LIN {X 0,Y 353.137,Z 586.014,A -85,B 0,C 180,E1 15983.414,E2 15983.414} C_VEL
LIN {X 0,Y 345.112,Z 562.488,A -85,B 0,C 180,E1 15988.238,E2 15988.238} C_VEL
LIN {X 0,Y 335.464,Z 541.503,A -85,B 0,C 180,E1 15993.705,E2 15993.705} C_VEL
LIN {X 0,Y 327.139,Z 526.718,A -85,B 0,C 180,E1 15998.911,E2 15998.911} C_VEL
LIN {X 0,Y 320.283,Z 515.167,A -85,B 0,C 180,E1 16004.452,E2 16004.452} C_VEL
LIN {X 0,Y 316.039,Z 508.566,A -85,B 0,C 180,E1 16009.304,E2 16009.304} C_VEL
LIN {X 0,Y 313.178,Z 504.462,A -85,B 0,C 180,E1 16018.617,E2 16018.617} C_VEL
LIN {X 0,Y 316.834,Z 509.857,A -85,B 0,C 180,E1 16027.466,E2 16027.466} C_VEL
LIN {X 0,Y 321.627,Z 517.983,A -85,B 0,C 180,E1 16032.576,E2 16032.576} C_VEL
LIN {X 0,Y 328.52,Z 529.301,A -85,B 0,C 180,E1 16037.778,E2 16037.778} C_VEL
LIN {X 0,Y 337.694,Z 547.182,A -85,B 0,C 180,E1 16043.535,E2 16043.535} C_VEL
LIN {X 0,Y 346.598,Z 568.688,A -85,B 0,C 180,E1 16048.719,E2 16048.719} C_VEL
LIN {X 0,Y 352.614,Z 590.285,A -85,B 0,C 180,E1 16052.83,E2 16052.83} C_VEL
LIN {X 0,Y 340.82,Z 629.242,A -85,B 0,C 180,E1 16055.81,E2 16055.81} C_VEL
LIN {X 0,Y 327.37,Z 665.336,A -85,B 0,C 180,E1 16059.799,E2 16059.799} C_VEL
LIN {X 0,Y 313.918,Z 696.935,A -85,B 0,C 180,E1 16064.711,E2 16064.711} C_VEL
LIN {X 0,Y 301.373,Z 724.654,A -85,B 0,C 180,E1 16070.701,E2 16070.701} C_VEL
LIN {X 0,Y 290.781,Z 748.154,A -85,B 0,C 180,E1 16077.768,E2 16077.768} C_VEL
LIN {X 0,Y 283.432,Z 766.757,A -85,B 0,C 180,E1 16085.741,E2 16085.741} C_VEL
LIN {X 0,Y 279.612,Z 780.048,A -85,B 0,C 180,E1 16094.291,E2 16094.291} C_VEL
LIN {X 0,Y 278.455,Z 786.164,A -85,B 0,C 180,E1 16100.611,E2 16100.611} C_VEL
LIN {X 0,Y 278.297,Z 789.212,A -85,B 0,C 180,E1 16106.881,E2 16106.881} C_VEL
LIN {X 0,Y 278.243,Z 789.212,A -85,B 0,C 180,E1 16113.119,E2 16113.119} C_VEL
LIN {X 0,Y 278.634,Z 785.021,A -85,B 0,C 180,E1 16120.802,E2 16120.802} C_VEL
LIN {X 0,Y 280.671,Z 775.811,A -85,B 0,C 180,E1 16128.886,E2 16128.886} C_VEL
LIN {X 0,Y 285.353,Z 761.575,A -85,B 0,C 180,E1 16136.809,E2 16136.809} C_VEL
LIN {X 0,Y 294.373,Z 740.19,A -85,B 0,C 180,E1 16144.905,E2 16144.905} C_VEL
LIN {X 0,Y 306.704,Z 712.859,A -85,B 0,C 180,E1 16152.112,E2 16152.112} C_VEL
LIN {X 0,Y 320.536,Z 682.014,A -85,B 0,C 180,E1 16157.82,E2 16157.82} C_VEL
LIN {X 0,Y 334.611,Z 647.007,A -85,B 0,C 180,E1 16162.409,E2 16162.409} C_VEL
LIN {X 0,Y 347.053,Z 610.454,A -85,B 0,C 180,E1 16165.773,E2 16165.773} C_VEL
LIN {X 0,Y 348.409,Z 599.608,A -85,B 0,C 180,E1 16166.985,E2 16166.985} C_VEL
LIN {X 0,Y 345.391,Z 584.533,A -85,B 0,C 180,E1 16169.727,E2 16169.727} C_VEL
LIN {X 0,Y 337.684,Z 561.735,A -85,B 0,C 180,E1 16174.828,E2 16174.828} C_VEL
LIN {X 0,Y 328.702,Z 541.555,A -85,B 0,C 180,E1 16180.754,E2 16180.754} C_VEL
LIN {X 0,Y 321.259,Z 528.092,A -85,B 0,C 180,E1 16186.457,E2 16186.457} C_VEL
LIN {X 0,Y 317.544,Z 522.011,A -85,B 0,C 180,E1 16190.046,E2 16190.046} C_VEL
LIN {X 0,Y 314.711,Z 516.201,A -85,B 0,C 180,E1 16194.131,E2 16194.131} C_VEL
LIN {X 0,Y 312.367,Z 513.05,A -85,B 0,C 180,E1 16199.998,E2 16199.998} C_VEL
LIN {X 0,Y 312.759,Z 514.467,A -85,B 0,C 180,E1 16206.251,E2 16206.251} C_VEL
LIN {X 0,Y 315.457,Z 517.712,A -85,B 0,C 180,E1 16211.31,E2 16211.31} C_VEL
LIN {X 0,Y 319.83,Z 525.512,A -85,B 0,C 180,E1 16216.411,E2 16216.411} C_VEL
LIN {X 0,Y 326.074,Z 535.896,A -85,B 0,C 180,E1 16221.437,E2 16221.437} C_VEL
LIN {X 0,Y 335.111,Z 553.88,A -85,B 0,C 180,E1 16227.401,E2 16227.401} C_VEL
LIN {X 0,Y 343.589,Z 575.487,A -85,B 0,C 180,E1 16232.717,E2 16232.717} C_VEL
LIN {X 0,Y 347.738,Z 591.04,A -85,B 0,C 180,E1 16235.805,E2 16235.805} C_VEL
LIN {X 0,Y 336.302,Z 626.527,A -85,B 0,C 180,E1 16238.531,E2 16238.531} C_VEL
LIN {X 0,Y 323.487,Z 658.718,A -85,B 0,C 180,E1 16242.125,E2 16242.125} C_VEL
LIN {X 0,Y 309.543,Z 688.272,A -85,B 0,C 180,E1 16246.779,E2 16246.779} C_VEL
LIN {X 0,Y 296.072,Z 714.128,A -85,B 0,C 180,E1 16252.606,E2 16252.606} C_VEL
LIN {X 0,Y 284.563,Z 735.641,A -85,B 0,C 180,E1 16259.636,E2 16259.636} C_VEL
LIN {X 0,Y 276.615,Z 751.803,A -85,B 0,C 180,E1 16267.47,E2 16267.47} C_VEL
LIN {X 0,Y 272.314,Z 762.47,A -85,B 0,C 180,E1 16275.51,E2 16275.51} C_VEL
LIN {X 0,Y 270.547,Z 768.232,A -85,B 0,C 180,E1 16283.573,E2 16283.573} C_VEL
LIN {X 0,Y 270.584,Z 769.634,A -85,B 0,C 180,E1 16290,E2 16290} C_VEL
LIN {X 0,Y 270.553,Z 768.178,A -85,B 0,C 180,E1 16296.427,E2 16296.427} C_VEL
LIN {X 0,Y 272.343,Z 762.375,A -85,B 0,C 180,E1 16304.489,E2 16304.489} C_VEL
LIN {X 0,Y 277.243,Z 750.314,A -85,B 0,C 180,E1 16313.325,E2 16313.325} C_VEL
LIN {X 0,Y 286.184,Z 732.442,A -85,B 0,C 180,E1 16321.498,E2 16321.498} C_VEL
LIN {X 0,Y 297.829,Z 710.843,A -85,B 0,C 180,E1 16328.155,E2 16328.155} C_VEL
LIN {X 0,Y 311.444,Z 684.319,A -85,B 0,C 180,E1 16333.851,E2 16333.851} C_VEL
LIN {X 0,Y 325.748,Z 653.106,A -85,B 0,C 180,E1 16338.516,E2 16338.516} C_VEL
LIN {X 0,Y 339.264,Z 617.956,A -85,B 0,C 180,E1 16342.129,E2 16342.129} C_VEL
LIN {X 0,Y 347.721,Z 589.37,A -85,B 0,C 180,E1 16344.295,E2 16344.295} C_VEL
LIN {X 0,Y 339.611,Z 564.718,A -85,B 0,C 180,E1 16349.644,E2 16349.644} C_VEL
LIN {X 0,Y 330.372,Z 544.154,A -85,B 0,C 180,E1 16355.464,E2 16355.464} C_VEL
LIN {X 0,Y 322.011,Z 528.726,A -85,B 0,C 180,E1 16361.536,E2 16361.536} C_VEL
LIN {X 0,Y 317.486,Z 521.686,A -85,B 0,C 180,E1 16365.708,E2 16365.708} C_VEL
LIN {X 0,Y 314.63,Z 516.234,A -85,B 0,C 180,E1 16369.65,E2 16369.65} C_VEL
LIN {X 0,Y 312.04,Z 512.261,A -85,B 0,C 180,E1 16378.611,E2 16378.611} C_VEL
LIN {X 0,Y 315.364,Z 517.62,A -85,B 0,C 180,E1 16387.241,E2 16387.241} C_VEL
LIN {X 0,Y 319.799,Z 525.722,A -85,B 0,C 180,E1 16392.388,E2 16392.388} C_VEL
LIN {X 0,Y 325.91,Z 536.494,A -85,B 0,C 180,E1 16397.402,E2 16397.402} C_VEL
LIN {X 0,Y 334.33,Z 553.843,A -85,B 0,C 180,E1 16403.098,E2 16403.098} C_VEL
LIN {X 0,Y 342.861,Z 576.373,A -85,B 0,C 180,E1 16408.609,E2 16408.609} C_VEL
LIN {X 0,Y 347.106,Z 593.898,A -85,B 0,C 180,E1 16411.983,E2 16411.983} C_VEL
LIN {X 0,Y 335.107,Z 631.506,A -85,B 0,C 180,E1 16414.94,E2 16414.94} C_VEL
LIN {X 0,Y 321.819,Z 665.824,A -85,B 0,C 180,E1 16418.808,E2 16418.808} C_VEL
LIN {X 0,Y 308.231,Z 696.335,A -85,B 0,C 180,E1 16423.57,E2 16423.57} C_VEL
LIN {X 0,Y 294.83,Z 724.689,A -85,B 0,C 180,E1 16429.787,E2 16429.787} C_VEL
LIN {X 0,Y 283.811,Z 747.971,A -85,B 0,C 180,E1 16436.937,E2 16436.937} C_VEL
LIN {X 0,Y 276.045,Z 766.29,A -85,B 0,C 180,E1 16444.966,E2 16444.966} C_VEL
LIN {X 0,Y 271.827,Z 779.746,A -85,B 0,C 180,E1 16453.829,E2 16453.829} C_VEL
LIN {X 0,Y 270.574,Z 785.87,A -85,B 0,C 180,E1 16460.335,E2 16460.335} C_VEL
LIN {X 0,Y 270.401,Z 788.924,A -85,B 0,C 180,E1 16466.79,E2 16466.79} C_VEL
LIN {X 0,Y 270.355,Z 788.925,A -85,B 0,C 180,E1 16473.21,E2 16473.21} C_VEL
LIN {X 0,Y 270.774,Z 784.86,A -85,B 0,C 180,E1 16480.953,E2 16480.953} C_VEL
LIN {X 0,Y 273,Z 775.452,A -85,B 0,C 180,E1 16489.476,E2 16489.476} C_VEL
LIN {X 0,Y 278.038,Z 761.26,A -85,B 0,C 180,E1 16497.574,E2 16497.574} C_VEL
LIN {X 0,Y 287.656,Z 739.855,A -85,B 0,C 180,E1 16505.844,E2 16505.844} C_VEL
LIN {X 0,Y 300.675,Z 712.5,A -85,B 0,C 180,E1 16513.159,E2 16513.159} C_VEL
LIN {X 0,Y 315.05,Z 681.606,A -85,B 0,C 180,E1 16518.933,E2 16518.933} C_VEL
LIN {X 0,Y 329.561,Z 646.887,A -85,B 0,C 180,E1 16523.495,E2 16523.495} C_VEL
LIN {X 0,Y 342.623,Z 609.563,A -85,B 0,C 180,E1 16526.92,E2 16526.92} C_VEL
LIN {X 0,Y 347.405,Z 592.925,A -85,B 0,C 180,E1 16528.102,E2 16528.102} C_VEL
LIN {X 0,Y 345.391,Z 584.533,A -85,B 0,C 180,E1 16529.727,E2 16529.727} C_VEL
LIN {X 0,Y 341.684,Z 578.36,A -85,B 0,C 180,E1 16531.557,E2 16531.557} C_VEL
LIN {X 0,Y 334.557,Z 569.967,A -85,B 0,C 180,E1 16534.821,E2 16534.821} C_VEL
LIN {X 0,Y 326.525,Z 550.443,A -85,B 0,C 180,E1 16540.532,E2 16540.532} C_VEL
LIN {X 0,Y 319.453,Z 536.042,A -85,B 0,C 180,E1 16546.379,E2 16546.379} C_VEL
LIN {X 0,Y 315.565,Z 529.312,A -85,B 0,C 180,E1 16550.506,E2 16550.506} C_VEL
LIN {X 0,Y 312.771,Z 523.658,A -85,B 0,C 180,E1 16554.791,E2 16554.791} C_VEL
LIN {X 0,Y 310.987,Z 520.863,A -85,B 0,C 180,E1 16559.998,E2 16559.998} C_VEL
LIN {X 0,Y 311.369,Z 522.333,A -85,B 0,C 180,E1 16566.371,E2 16566.371} C_VEL
LIN {X 0,Y 313.758,Z 525.368,A -85,B 0,C 180,E1 16571.064,E2 16571.064} C_VEL
LIN {X 0,Y 317.849,Z 533.119,A -85,B 0,C 180,E1 16576.165,E2 16576.165} C_VEL
LIN {X 0,Y 323.837,Z 543.834,A -85,B 0,C 180,E1 16581.317,E2 16581.317} C_VEL
LIN {X 0,Y 331.922,Z 561.078,A -85,B 0,C 180,E1 16587.135,E2 16587.135} C_VEL
LIN {X 0,Y 339.909,Z 583.609,A -85,B 0,C 180,E1 16592.711,E2 16592.711} C_VEL
LIN {X 0,Y 342.528,Z 593.61,A -85,B 0,C 180,E1 16594.827,E2 16594.827} C_VEL
LIN {X 0,Y 329.727,Z 631.56,A -85,B 0,C 180,E1 16597.883,E2 16597.883} C_VEL
LIN {X 0,Y 314.704,Z 666.624,A -85,B 0,C 180,E1 16602.078,E2 16602.078} C_VEL
LIN {X 0,Y 299.679,Z 696.377,A -85,B 0,C 180,E1 16607.288,E2 16607.288} C_VEL
LIN {X 0,Y 285.425,Z 722.099,A -85,B 0,C 180,E1 16613.879,E2 16613.879} C_VEL
LIN {X 0,Y 274.858,Z 741.051,A -85,B 0,C 180,E1 16620.971,E2 16620.971} C_VEL
LIN {X 0,Y 267.351,Z 755.919,A -85,B 0,C 180,E1 16629.316,E2 16629.316} C_VEL
LIN {X 0,Y 263.877,Z 764.691,A -85,B 0,C 180,E1 16637.243,E2 16637.243} C_VEL
LIN {X 0,Y 262.664,Z 768.521,A -85,B 0,C 180,E1 16643.38,E2 16643.38} C_VEL
LIN {X 0,Y 262.684,Z 769.921,A -85,B 0,C 180,E1 16650,E2 16650} C_VEL
LIN {X 0,Y 262.671,Z 768.468,A -85,B 0,C 180,E1 16656.62,E2 16656.62} C_VEL
LIN {X 0,Y 264.602,Z 762.668,A -85,B 0,C 180,E1 16664.922,E2 16664.922} C_VEL
LIN {X 0,Y 269.839,Z 750.62,A -85,B 0,C 180,E1 16674.005,E2 16674.005} C_VEL
LIN {X 0,Y 279.318,Z 732.761,A -85,B 0,C 180,E1 16682.365,E2 16682.365} C_VEL
LIN {X 0,Y 292.134,Z 710.066,A -85,B 0,C 180,E1 16689.414,E2 16689.414} C_VEL
LIN {X 0,Y 306.658,Z 682.818,A -85,B 0,C 180,E1 16695.216,E2 16695.216} C_VEL
LIN {X 0,Y 321.286,Z 651.843,A -85,B 0,C 180,E1 16699.78,E2 16699.78} C_VEL
LIN {X 0,Y 335.034,Z 616.822,A -85,B 0,C 180,E1 16703.339,E2 16703.339} C_VEL
LIN {X 0,Y 342.454,Z 593.221,A -85,B 0,C 180,E1 16705.119,E2 16705.119} C_VEL
LIN {X 0,Y 335.089,Z 569.345,A -85,B 0,C 180,E1 16710.535,E2 16710.535} C_VEL
LIN {X 0,Y 326.861,Z 550.145,A -85,B 0,C 180,E1 16716.184,E2 16716.184} C_VEL
LIN {X 0,Y 319.519,Z 535.81,A -85,B 0,C 180,E1 16722.045,E2 16722.045} C_VEL
LIN {X 0,Y 315.478,Z 528.945,A -85,B 0,C 180,E1 16726.216,E2 16726.216} C_VEL
LIN {X 0,Y 312.922,Z 523.837,A -85,B 0,C 180,E1 16729.968,E2 16729.968} C_VEL
LIN {X 0,Y 310.706,Z 520.048,A -85,B 0,C 180,E1 16738.606,E2 16738.606} C_VEL
LIN {X 0,Y 313.615,Z 525.144,A -85,B 0,C 180,E1 16746.933,E2 16746.933} C_VEL
LIN {X 0,Y 317.885,Z 533.565,A -85,B 0,C 180,E1 16752.29,E2 16752.29} C_VEL
LIN {X 0,Y 323.985,Z 545.148,A -85,B 0,C 180,E1 16757.592,E2 16757.592} C_VEL
LIN {X 0,Y 331.143,Z 561.142,A -85,B 0,C 180,E1 16762.861,E2 16762.861} C_VEL
LIN {X 0,Y 338.456,Z 582.174,A -85,B 0,C 180,E1 16768.102,E2 16768.102} C_VEL
LIN {X 0,Y 341.793,Z 597.172,A -85,B 0,C 180,E1 16771.093,E2 16771.093} C_VEL
LIN {X 0,Y 327.694,Z 638.464,A -85,B 0,C 180,E1 16774.49,E2 16774.49} C_VEL
LIN {X 0,Y 312.596,Z 674.634,A -85,B 0,C 180,E1 16778.92,E2 16778.92} C_VEL
LIN {X 0,Y 297.477,Z 706.575,A -85,B 0,C 180,E1 16784.554,E2 16784.554} C_VEL
LIN {X 0,Y 283.977,Z 733.239,A -85,B 0,C 180,E1 16791.208,E2 16791.208} C_VEL
LIN {X 0,Y 272.971,Z 755.957,A -85,B 0,C 180,E1 16799.373,E2 16799.373} C_VEL
LIN {X 0,Y 266.107,Z 772.766,A -85,B 0,C 180,E1 16808.294,E2 16808.294} C_VEL
LIN {X 0,Y 263.218,Z 782.902,A -85,B 0,C 180,E1 16816.697,E2 16816.697} C_VEL
LIN {X 0,Y 262.421,Z 787.482,A -85,B 0,C 180,E1 16823.373,E2 16823.373} C_VEL
LIN {X 0,Y 262.646,Z 789.025,A -85,B 0,C 180,E1 16830,E2 16830} C_VEL
LIN {X 0,Y 262.426,Z 787.489,A -85,B 0,C 180,E1 16836.626,E2 16836.626} C_VEL
LIN {X 0,Y 263.606,Z 781.259,A -85,B 0,C 180,E1 16844.98,E2 16844.98} C_VEL
LIN {X 0,Y 267.024,Z 770.117,A -85,B 0,C 180,E1 16853.386,E2 16853.386} C_VEL
LIN {X 0,Y 274.247,Z 753.319,A -85,B 0,C 180,E1 16861.755,E2 16861.755} C_VEL
LIN {X 0,Y 285.355,Z 730.673,A -85,B 0,C 180,E1 16869.549,E2 16869.549} C_VEL
LIN {X 0,Y 299.435,Z 702.663,A -85,B 0,C 180,E1 16876.269,E2 16876.269} C_VEL
LIN {X 0,Y 314.667,Z 670.229,A -85,B 0,C 180,E1 16881.715,E2 16881.715} C_VEL
LIN {X 0,Y 329.211,Z 634.734,A -85,B 0,C 180,E1 16885.881,E2 16885.881} C_VEL
LIN {X 0,Y 342.019,Z 596.191,A -85,B 0,C 180,E1 16889.016,E2 16889.016} C_VEL
LIN {X 0,Y 335.616,Z 572.905,A -85,B 0,C 180,E1 16894.076,E2 16894.076} C_VEL
LIN {X 0,Y 334.557,Z 569.967,A -85,B 0,C 180,E1 16894.821,E2 16894.821} C_VEL
LIN {X 0,Y 330.732,Z 565.067,A -85,B 0,C 180,E1 16896.813,E2 16896.813} C_VEL
LIN {X 0,Y 324.612,Z 559.901,A -85,B 0,C 180,E1 16900.015,E2 16900.015} C_VEL
LIN {X 0,Y 324.191,Z 558.921,A -85,B 0,C 180,E1 16900.358,E2 16900.358} C_VEL
LIN {X 0,Y 317.096,Z 543.325,A -85,B 0,C 180,E1 16906.721,E2 16906.721} C_VEL
LIN {X 0,Y 313.157,Z 536.373,A -85,B 0,C 180,E1 16911.134,E2 16911.134} C_VEL
LIN {X 0,Y 311.193,Z 531.423,A -85,B 0,C 180,E1 16914.765,E2 16914.765} C_VEL
LIN {X 0,Y 309.487,Z 528.638,A -85,B 0,C 180,E1 16919.998,E2 16919.998} C_VEL
LIN {X 0,Y 309.811,Z 530.002,A -85,B 0,C 180,E1 16926.189,E2 16926.189} C_VEL
LIN {X 0,Y 311.916,Z 532.916,A -85,B 0,C 180,E1 16930.77,E2 16930.77} C_VEL
LIN {X 0,Y 315.728,Z 540.724,A -85,B 0,C 180,E1 16935.978,E2 16935.978} C_VEL
LIN {X 0,Y 321.027,Z 551.025,A -85,B 0,C 180,E1 16940.983,E2 16940.983} C_VEL
LIN {X 0,Y 328.008,Z 566.848,A -85,B 0,C 180,E1 16946.464,E2 16946.464} C_VEL
LIN {X 0,Y 335.297,Z 589.367,A -85,B 0,C 180,E1 16952.222,E2 16952.222} C_VEL
LIN {X 0,Y 336.939,Z 598.552,A -85,B 0,C 180,E1 16954.062,E2 16954.062} C_VEL
LIN {X 0,Y 323.756,Z 634.87,A -85,B 0,C 180,E1 16957.063,E2 16957.063} C_VEL
LIN {X 0,Y 308.734,Z 668.307,A -85,B 0,C 180,E1 16961.174,E2 16961.174} C_VEL
LIN {X 0,Y 293.399,Z 697.437,A -85,B 0,C 180,E1 16966.381,E2 16966.381} C_VEL
LIN {X 0,Y 279.454,Z 721.6,A -85,B 0,C 180,E1 16972.64,E2 16972.64} C_VEL
LIN {X 0,Y 267.915,Z 741.21,A -85,B 0,C 180,E1 16980.062,E2 16980.062} C_VEL
LIN {X 0,Y 259.727,Z 756.417,A -85,B 0,C 180,E1 16988.845,E2 16988.845} C_VEL
LIN {X 0,Y 256.244,Z 764.534,A -85,B 0,C 180,E1 16996.328,E2 16996.328} C_VEL
LIN {X 0,Y 254.782,Z 768.809,A -85,B 0,C 180,E1 17003.174,E2 17003.174} C_VEL
LIN {X 0,Y 254.802,Z 770.208,A -85,B 0,C 180,E1 17010,E2 17010} C_VEL
LIN {X 0,Y 254.79,Z 768.757,A -85,B 0,C 180,E1 17016.826,E2 17016.826} C_VEL
LIN {X 0,Y 256.851,Z 762.961,A -85,B 0,C 180,E1 17025.383,E2 17025.383} C_VEL
LIN {X 0,Y 262.503,Z 750.924,A -85,B 0,C 180,E1 17034.72,E2 17034.72} C_VEL
LIN {X 0,Y 272.538,Z 733.077,A -85,B 0,C 180,E1 17043.273,E2 17043.273} C_VEL
LIN {X 0,Y 285.949,Z 710.405,A -85,B 0,C 180,E1 17050.44,E2 17050.44} C_VEL
LIN {X 0,Y 301.066,Z 683.188,A -85,B 0,C 180,E1 17056.299,E2 17056.299} C_VEL
LIN {X 0,Y 316.129,Z 652.423,A -85,B 0,C 180,E1 17060.866,E2 17060.866} C_VEL
LIN {X 0,Y 330.369,Z 617.365,A -85,B 0,C 180,E1 17064.441,E2 17064.441} C_VEL
LIN {X 0,Y 337.064,Z 597.828,A -85,B 0,C 180,E1 17065.891,E2 17065.891} C_VEL
LIN {X 0,Y 332.03,Z 578.634,A -85,B 0,C 180,E1 17070.237,E2 17070.237} C_VEL
LIN {X 0,Y 324.684,Z 558.924,A -85,B 0,C 180,E1 17075.922,E2 17075.922} C_VEL
LIN {X 0,Y 317.28,Z 543.256,A -85,B 0,C 180,E1 17082.301,E2 17082.301} C_VEL
LIN {X 0,Y 313.251,Z 536.151,A -85,B 0,C 180,E1 17086.702,E2 17086.702} C_VEL
LIN {X 0,Y 311.15,Z 531.459,A -85,B 0,C 180,E1 17090.286,E2 17090.286} C_VEL
LIN {X 0,Y 309.213,Z 527.806,A -85,B 0,C 180,E1 17098.599,E2 17098.599} C_VEL
LIN {X 0,Y 311.766,Z 532.824,A -85,B 0,C 180,E1 17106.712,E2 17106.712} C_VEL
LIN {X 0,Y 315.732,Z 541.197,A -85,B 0,C 180,E1 17112.111,E2 17112.111} C_VEL
LIN {X 0,Y 322.296,Z 554.591,A -85,B 0,C 180,E1 17118.19,E2 17118.19} C_VEL
LIN {X 0,Y 330.026,Z 574.809,A -85,B 0,C 180,E1 17124.386,E2 17124.386} C_VEL
LIN {X 0,Y 336.228,Z 597.696,A -85,B 0,C 180,E1 17129.691,E2 17129.691} C_VEL
LIN {X 0,Y 335.819,Z 602.485,A -85,B 0,C 180,E1 17130.332,E2 17130.332} C_VEL
LIN {X 0,Y 322.438,Z 639.685,A -85,B 0,C 180,E1 17133.474,E2 17133.474} C_VEL
LIN {X 0,Y 306.978,Z 675.305,A -85,B 0,C 180,E1 17137.891,E2 17137.891} C_VEL
LIN {X 0,Y 291.715,Z 706.212,A -85,B 0,C 180,E1 17143.392,E2 17143.392} C_VEL
LIN {X 0,Y 277.403,Z 733.23,A -85,B 0,C 180,E1 17150.24,E2 17150.24} C_VEL
LIN {X 0,Y 266.226,Z 755.026,A -85,B 0,C 180,E1 17158.185,E2 17158.185} C_VEL
LIN {X 0,Y 258.962,Z 771.185,A -85,B 0,C 180,E1 17166.755,E2 17166.755} C_VEL
LIN {X 0,Y 255.816,Z 780.95,A -85,B 0,C 180,E1 17174.553,E2 17174.553} C_VEL
LIN {X 0,Y 254.537,Z 787.192,A -85,B 0,C 180,E1 17183.167,E2 17183.167} C_VEL
LIN {X 0,Y 254.768,Z 788.739,A -85,B 0,C 180,E1 17190,E2 17190} C_VEL
LIN {X 0,Y 254.542,Z 787.199,A -85,B 0,C 180,E1 17196.833,E2 17196.833} C_VEL
LIN {X 0,Y 255.815,Z 780.963,A -85,B 0,C 180,E1 17205.447,E2 17205.447} C_VEL
LIN {X 0,Y 259.513,Z 769.809,A -85,B 0,C 180,E1 17214.105,E2 17214.105} C_VEL
LIN {X 0,Y 267.13,Z 753.13,A -85,B 0,C 180,E1 17222.64,E2 17222.64} C_VEL
LIN {X 0,Y 279.006,Z 730.332,A -85,B 0,C 180,E1 17230.634,E2 17230.634} C_VEL
LIN {X 0,Y 293.95,Z 701.944,A -85,B 0,C 180,E1 17237.504,E2 17237.504} C_VEL
LIN {X 0,Y 309.645,Z 669.808,A -85,B 0,C 180,E1 17242.908,E2 17242.908} C_VEL
LIN {X 0,Y 324.741,Z 634.232,A -85,B 0,C 180,E1 17247.063,E2 17247.063} C_VEL
LIN {X 0,Y 336.639,Z 599.376,A -85,B 0,C 180,E1 17249.978,E2 17249.978} C_VEL
LIN {X 0,Y 331.372,Z 578.764,A -85,B 0,C 180,E1 17254.618,E2 17254.618} C_VEL
LIN {X 0,Y 324.191,Z 558.921,A -85,B 0,C 180,E1 17260.358,E2 17260.358} C_VEL
LIN {X 0,Y 320.766,Z 555.603,A -85,B 0,C 180,E1 17262.536,E2 17262.536} C_VEL
LIN {X 0,Y 315.39,Z 552.897,A -85,B 0,C 180,E1 17265.975,E2 17265.975} C_VEL
LIN {X 0,Y 315.066,Z 552.056,A -85,B 0,C 180,E1 17266.343,E2 17266.343} C_VEL
LIN {X 0,Y 311.27,Z 544.188,A -85,B 0,C 180,E1 17271.08,E2 17271.08} C_VEL
LIN {X 0,Y 308.977,Z 538.755,A -85,B 0,C 180,E1 17275.432,E2 17275.432} C_VEL
LIN {X 0,Y 307.692,Z 536.354,A -85,B 0,C 180,E1 17279.998,E2 17279.998} C_VEL
LIN {X 0,Y 307.932,Z 537.6,A -85,B 0,C 180,E1 17286.012,E2 17286.012} C_VEL
LIN {X 0,Y 309.883,Z 540.498,A -85,B 0,C 180,E1 17290.522,E2 17290.522} C_VEL
LIN {X 0,Y 313.385,Z 548.242,A -85,B 0,C 180,E1 17295.765,E2 17295.765} C_VEL
LIN {X 0,Y 318.425,Z 558.829,A -85,B 0,C 180,E1 17300.889,E2 17300.889} C_VEL
LIN {X 0,Y 324.355,Z 573.435,A -85,B 0,C 180,E1 17306.039,E2 17306.039} C_VEL
LIN {X 0,Y 330.746,Z 595.28,A -85,B 0,C 180,E1 17311.761,E2 17311.761} C_VEL
LIN {X 0,Y 331.855,Z 601.305,A -85,B 0,C 180,E1 17313.087,E2 17313.087} C_VEL
LIN {X 0,Y 318.442,Z 636.689,A -85,B 0,C 180,E1 17316.068,E2 17316.068} C_VEL
LIN {X 0,Y 303.353,Z 669.041,A -85,B 0,C 180,E1 17320.095,E2 17320.095} C_VEL
LIN {X 0,Y 287.64,Z 697.774,A -85,B 0,C 180,E1 17325.278,E2 17325.278} C_VEL
LIN {X 0,Y 272.876,Z 722.214,A -85,B 0,C 180,E1 17331.707,E2 17331.707} C_VEL
LIN {X 0,Y 260.602,Z 742.052,A -85,B 0,C 180,E1 17339.445,E2 17339.445} C_VEL
LIN {X 0,Y 252.248,Z 756.711,A -85,B 0,C 180,E1 17348.186,E2 17348.186} C_VEL
LIN {X 0,Y 248.01,Z 766.142,A -85,B 0,C 180,E1 17357.599,E2 17357.599} C_VEL
LIN {X 0,Y 246.734,Z 770.155,A -85,B 0,C 180,E1 17366.482,E2 17366.482} C_VEL
LIN {X 0,Y 246.751,Z 770.124,A -85,B 0,C 180,E1 17373.518,E2 17373.518} C_VEL
LIN {X 0,Y 248.033,Z 766.054,A -85,B 0,C 180,E1 17382.425,E2 17382.425} C_VEL
LIN {X 0,Y 252.307,Z 756.528,A -85,B 0,C 180,E1 17391.849,E2 17391.849} C_VEL
LIN {X 0,Y 260.701,Z 741.816,A -85,B 0,C 180,E1 17400.565,E2 17400.565} C_VEL
LIN {X 0,Y 274.092,Z 720.165,A -85,B 0,C 180,E1 17408.846,E2 17408.846} C_VEL
LIN {X 0,Y 289.761,Z 693.948,A -85,B 0,C 180,E1 17415.433,E2 17415.433} C_VEL
LIN {X 0,Y 306.053,Z 663.415,A -85,B 0,C 180,E1 17420.624,E2 17420.624} C_VEL
LIN {X 0,Y 321.023,Z 630.34,A -85,B 0,C 180,E1 17424.45,E2 17424.45} C_VEL
LIN {X 0,Y 331.793,Z 600.108,A -85,B 0,C 180,E1 17426.998,E2 17426.998} C_VEL
LIN {X 0,Y 326.001,Z 578.645,A -85,B 0,C 180,E1 17432.33,E2 17432.33} C_VEL
LIN {X 0,Y 319.718,Z 561.77,A -85,B 0,C 180,E1 17437.741,E2 17437.741} C_VEL
LIN {X 0,Y 313.606,Z 548.705,A -85,B 0,C 180,E1 17443.734,E2 17443.734} C_VEL
LIN {X 0,Y 310.836,Z 543.113,A -85,B 0,C 180,E1 17447.395,E2 17447.395} C_VEL
LIN {X 0,Y 309.044,Z 538.926,A -85,B 0,C 180,E1 17450.724,E2 17450.724} C_VEL
LIN {X 0,Y 307.469,Z 535.482,A -85,B 0,C 180,E1 17458.591,E2 17458.591} C_VEL
LIN {X 0,Y 309.742,Z 540.392,A -85,B 0,C 180,E1 17466.492,E2 17466.492} C_VEL
LIN {X 0,Y 313.817,Z 549.6,A -85,B 0,C 180,E1 17472.452,E2 17472.452} C_VEL
LIN {X 0,Y 319.405,Z 562.422,A -85,B 0,C 180,E1 17478.089,E2 17478.089} C_VEL
LIN {X 0,Y 326.051,Z 581.254,A -85,B 0,C 180,E1 17483.974,E2 17483.974} C_VEL
LIN {X 0,Y 331.097,Z 601.956,A -85,B 0,C 180,E1 17488.936,E2 17488.936} C_VEL
LIN {X 0,Y 330.348,Z 606.289,A -85,B 0,C 180,E1 17489.442,E2 17489.442} C_VEL
LIN {X 0,Y 316.103,Z 643.756,A -85,B 0,C 180,E1 17492.728,E2 17492.728} C_VEL
LIN {X 0,Y 300.57,Z 677.734,A -85,B 0,C 180,E1 17497.088,E2 17497.088} C_VEL
LIN {X 0,Y 285.259,Z 707.355,A -85,B 0,C 180,E1 17502.519,E2 17502.519} C_VEL
LIN {X 0,Y 270.314,Z 734.237,A -85,B 0,C 180,E1 17509.549,E2 17509.549} C_VEL
LIN {X 0,Y 259.122,Z 754.847,A -85,B 0,C 180,E1 17517.282,E2 17517.282} C_VEL
LIN {X 0,Y 251.438,Z 770.875,A -85,B 0,C 180,E1 17526.016,E2 17526.016} C_VEL
LIN {X 0,Y 248.035,Z 780.653,A -85,B 0,C 180,E1 17534.056,E2 17534.056} C_VEL
LIN {X 0,Y 246.632,Z 786.901,A -85,B 0,C 180,E1 17542.947,E2 17542.947} C_VEL
LIN {X 0,Y 246.866,Z 788.451,A -85,B 0,C 180,E1 17550,E2 17550} C_VEL
LIN {X 0,Y 246.638,Z 786.909,A -85,B 0,C 180,E1 17557.053,E2 17557.053} C_VEL
LIN {X 0,Y 248.034,Z 780.667,A -85,B 0,C 180,E1 17565.944,E2 17565.944} C_VEL
LIN {X 0,Y 252.036,Z 769.502,A -85,B 0,C 180,E1 17574.868,E2 17574.868} C_VEL
LIN {X 0,Y 260.107,Z 752.936,A -85,B 0,C 180,E1 17583.574,E2 17583.574} C_VEL
LIN {X 0,Y 272.793,Z 729.994,A -85,B 0,C 180,E1 17591.764,E2 17591.764} C_VEL
LIN {X 0,Y 288.133,Z 702.186,A -85,B 0,C 180,E1 17598.589,E2 17598.589} C_VEL
LIN {X 0,Y 304.219,Z 670.568,A -85,B 0,C 180,E1 17603.977,E2 17603.977} C_VEL
LIN {X 0,Y 319.79,Z 635.289,A -85,B 0,C 180,E1 17608.136,E2 17608.136} C_VEL
LIN {X 0,Y 331.398,Z 603.562,A -85,B 0,C 180,E1 17610.751,E2 17610.751} C_VEL
LIN {X 0,Y 326.346,Z 582.066,A -85,B 0,C 180,E1 17615.851,E2 17615.851} C_VEL
LIN {X 0,Y 319.397,Z 562.07,A -85,B 0,C 180,E1 17622.066,E2 17622.066} C_VEL
LIN {X 0,Y 315.066,Z 552.056,A -85,B 0,C 180,E1 17626.343,E2 17626.343} C_VEL
LIN {X 0,Y 313.118,Z 551.062,A -85,B 0,C 180,E1 17627.879,E2 17627.879} C_VEL
LIN {X 0,Y 309.401,Z 552.394,A -85,B 0,C 180,E1 17630.566,E2 17630.566} C_VEL
LIN {X 0,Y 306.846,Z 546.241,A -85,B 0,C 180,E1 17635.754,E2 17635.754} C_VEL
LIN {X 0,Y 305.711,Z 543.87,A -85,B 0,C 180,E1 17642.837,E2 17642.837} C_VEL
LIN {X 0,Y 307.702,Z 548.113,A -85,B 0,C 180,E1 17650.347,E2 17650.347} C_VEL
LIN {X 0,Y 311.109,Z 556.094,A -85,B 0,C 180,E1 17655.794,E2 17655.794} C_VEL
LIN {X 0,Y 316.58,Z 568.715,A -85,B 0,C 180,E1 17661.752,E2 17661.752} C_VEL
LIN {X 0,Y 322.564,Z 586.776,A -85,B 0,C 180,E1 17667.6,E2 17667.6} C_VEL
LIN {X 0,Y 326.677,Z 604.352,A -85,B 0,C 180,E1 17672.076,E2 17672.076} C_VEL
LIN {X 0,Y 312.287,Z 640.625,A -85,B 0,C 180,E1 17675.261,E2 17675.261} C_VEL
LIN {X 0,Y 296.493,Z 672.735,A -85,B 0,C 180,E1 17679.43,E2 17679.43} C_VEL
LIN {X 0,Y 280.378,Z 700.708,A -85,B 0,C 180,E1 17684.71,E2 17684.71} C_VEL
LIN {X 0,Y 265.557,Z 724.094,A -85,B 0,C 180,E1 17691.157,E2 17691.157} C_VEL
LIN {X 0,Y 253.668,Z 742.352,A -85,B 0,C 180,E1 17698.514,E2 17698.514} C_VEL
LIN {X 0,Y 244.956,Z 756.745,A -85,B 0,C 180,E1 17707.274,E2 17707.274} C_VEL
LIN {X 0,Y 240.207,Z 766.432,A -85,B 0,C 180,E1 17717.189,E2 17717.189} C_VEL
LIN {X 0,Y 238.831,Z 770.443,A -85,B 0,C 180,E1 17726.365,E2 17726.365} C_VEL
LIN {X 0,Y 238.848,Z 770.412,A -85,B 0,C 180,E1 17733.635,E2 17733.635} C_VEL
LIN {X 0,Y 240.232,Z 766.345,A -85,B 0,C 180,E1 17742.836,E2 17742.836} C_VEL
LIN {X 0,Y 244.978,Z 756.613,A -85,B 0,C 180,E1 17752.724,E2 17752.724} C_VEL
LIN {X 0,Y 254.882,Z 740.414,A -85,B 0,C 180,E1 17762.32,E2 17762.32} C_VEL
LIN {X 0,Y 268.532,Z 719.414,A -85,B 0,C 180,E1 17770.249,E2 17770.249} C_VEL
LIN {X 0,Y 284.733,Z 693.397,A -85,B 0,C 180,E1 17776.764,E2 17776.764} C_VEL
LIN {X 0,Y 301.059,Z 663.813,A -85,B 0,C 180,E1 17781.798,E2 17781.798} C_VEL
LIN {X 0,Y 316.472,Z 630.837,A -85,B 0,C 180,E1 17785.62,E2 17785.62} C_VEL
LIN {X 0,Y 326.568,Z 603.902,A -85,B 0,C 180,E1 17787.899,E2 17787.899} C_VEL
LIN {X 0,Y 321.096,Z 582.134,A -85,B 0,C 180,E1 17793.631,E2 17793.631} C_VEL
LIN {X 0,Y 314.953,Z 565.021,A -85,B 0,C 180,E1 17799.606,E2 17799.606} C_VEL
LIN {X 0,Y 309.449,Z 552.09,A -85,B 0,C 180,E1 17806.269,E2 17806.269} C_VEL
LIN {X 0,Y 306.901,Z 546.456,A -85,B 0,C 180,E1 17811.034,E2 17811.034} C_VEL
LIN {X 0,Y 305.631,Z 543.144,A -85,B 0,C 180,E1 17818.582,E2 17818.582} C_VEL
LIN {X 0,Y 307.524,Z 547.976,A -85,B 0,C 180,E1 17826.292,E2 17826.292} C_VEL
LIN {X 0,Y 311.226,Z 556.884,A -85,B 0,C 180,E1 17832.156,E2 17832.156} C_VEL
LIN {X 0,Y 316.321,Z 569.755,A -85,B 0,C 180,E1 17837.875,E2 17837.875} C_VEL
LIN {X 0,Y 322.277,Z 588.941,A -85,B 0,C 180,E1 17843.904,E2 17843.904} C_VEL
LIN {X 0,Y 326.03,Z 606.464,A -85,B 0,C 180,E1 17848.215,E2 17848.215} C_VEL
LIN {X 0,Y 311.769,Z 643.281,A -85,B 0,C 180,E1 17851.467,E2 17851.467} C_VEL
LIN {X 0,Y 295.52,Z 677.685,A -85,B 0,C 180,E1 17855.875,E2 17855.875} C_VEL
LIN {X 0,Y 279.661,Z 707.141,A -85,B 0,C 180,E1 17861.304,E2 17861.304} C_VEL
LIN {X 0,Y 264.845,Z 732.705,A -85,B 0,C 180,E1 17868.001,E2 17868.001} C_VEL
LIN {X 0,Y 252.185,Z 754.531,A -85,B 0,C 180,E1 17876.263,E2 17876.263} C_VEL
LIN {X 0,Y 243.969,Z 770.567,A -85,B 0,C 180,E1 17885.233,E2 17885.233} C_VEL
LIN {X 0,Y 240.258,Z 780.355,A -85,B 0,C 180,E1 17893.525,E2 17893.525} C_VEL
LIN {X 0,Y 238.756,Z 786.611,A -85,B 0,C 180,E1 17902.713,E2 17902.713} C_VEL
LIN {X 0,Y 238.994,Z 788.165,A -85,B 0,C 180,E1 17910,E2 17910} C_VEL
LIN {X 0,Y 238.762,Z 786.62,A -85,B 0,C 180,E1 17917.286,E2 17917.286} C_VEL
LIN {X 0,Y 240.255,Z 780.37,A -85,B 0,C 180,E1 17926.475,E2 17926.475} C_VEL
LIN {X 0,Y 244.604,Z 769.196,A -85,B 0,C 180,E1 17935.678,E2 17935.678} C_VEL
LIN {X 0,Y 253.254,Z 752.617,A -85,B 0,C 180,E1 17944.609,E2 17944.609} C_VEL
LIN {X 0,Y 266.672,Z 729.658,A -85,B 0,C 180,E1 17952.949,E2 17952.949} C_VEL
LIN {X 0,Y 282.136,Z 702.935,A -85,B 0,C 180,E1 17959.621,E2 17959.621} C_VEL
LIN {X 0,Y 299.359,Z 670.384,A -85,B 0,C 180,E1 17965.214,E2 17965.214} C_VEL
LIN {X 0,Y 315.548,Z 634.787,A -85,B 0,C 180,E1 17969.397,E2 17969.397} C_VEL
LIN {X 0,Y 326.116,Z 606.555,A -85,B 0,C 180,E1 17971.787,E2 17971.787} C_VEL
LIN {X 0,Y 321.417,Z 585.387,A -85,B 0,C 180,E1 17977.131,E2 17977.131} C_VEL
LIN {X 0,Y 315.355,Z 566.855,A -85,B 0,C 180,E1 17983.257,E2 17983.257} C_VEL
LIN {X 0,Y 309.639,Z 552.65,A -85,B 0,C 180,E1 17990.284,E2 17990.284} C_VEL
LIN {X 0,Y 309.401,Z 552.394,A -85,B 0,C 180,E1 17990.566,E2 17990.566} C_VEL
LIN {X 0,Y 306.358,Z 552.475,A -85,B 0,C 180,E1 17993.804,E2 17993.804} C_VEL
LIN {X 0,Y 304.132,Z 553.158,A -85,B 0,C 180,E1 17997.11,E2 17997.11} C_VEL
LIN {X 0,Y 303.528,Z 551.479,A -85,B 0,C 180,E1 18002.857,E2 18002.857} C_VEL
LIN {X 0,Y 305.361,Z 555.593,A -85,B 0,C 180,E1 18010.125,E2 18010.125} C_VEL
LIN {X 0,Y 309.515,Z 565.994,A -85,B 0,C 180,E1 18017.065,E2 18017.065} C_VEL
LIN {X 0,Y 315.141,Z 581.53,A -85,B 0,C 180,E1 18023.558,E2 18023.558} C_VEL
LIN {X 0,Y 320.229,Z 601.006,A -85,B 0,C 180,E1 18029.372,E2 18029.372} C_VEL
LIN {X 0,Y 321.445,Z 607.526,A -85,B 0,C 180,E1 18031.006,E2 18031.006} C_VEL
LIN {X 0,Y 305.979,Z 644.982,A -85,B 0,C 180,E1 18034.465,E2 18034.465} C_VEL
LIN {X 0,Y 288.941,Z 677.725,A -85,B 0,C 180,E1 18038.956,E2 18038.956} C_VEL
LIN {X 0,Y 271.634,Z 706.042,A -85,B 0,C 180,E1 18044.708,E2 18044.708} C_VEL
LIN {X 0,Y 255.472,Z 730.052,A -85,B 0,C 180,E1 18052.055,E2 18052.055} C_VEL
LIN {X 0,Y 242.681,Z 748.729,A -85,B 0,C 180,E1 18060.85,E2 18060.85} C_VEL
LIN {X 0,Y 235.492,Z 760.651,A -85,B 0,C 180,E1 18069.635,E2 18069.635} C_VEL
LIN {X 0,Y 231.921,Z 767.904,A -85,B 0,C 180,E1 18078.705,E2 18078.705} C_VEL
LIN {X 0,Y 230.929,Z 770.731,A -85,B 0,C 180,E1 18086.241,E2 18086.241} C_VEL
LIN {X 0,Y 230.946,Z 770.701,A -85,B 0,C 180,E1 18093.759,E2 18093.759} C_VEL
LIN {X 0,Y 232.442,Z 766.647,A -85,B 0,C 180,E1 18103.257,E2 18103.257} C_VEL
LIN {X 0,Y 237.562,Z 756.909,A -85,B 0,C 180,E1 18113.475,E2 18113.475} C_VEL
LIN {X 0,Y 248.076,Z 740.724,A -85,B 0,C 180,E1 18123.32,E2 18123.32} C_VEL
LIN {X 0,Y 262.623,Z 719.473,A -85,B 0,C 180,E1 18131.463,E2 18131.463} C_VEL
LIN {X 0,Y 279.621,Z 693.226,A -85,B 0,C 180,E1 18138.066,E2 18138.066} C_VEL
LIN {X 0,Y 296.209,Z 664.216,A -85,B 0,C 180,E1 18143.007,E2 18143.007} C_VEL
LIN {X 0,Y 312.705,Z 629.812,A -85,B 0,C 180,E1 18146.959,E2 18146.959} C_VEL
LIN {X 0,Y 321.437,Z 607.85,A -85,B 0,C 180,E1 18148.797,E2 18148.797} C_VEL
LIN {X 0,Y 316.675,Z 587.008,A -85,B 0,C 180,E1 18154.517,E2 18154.517} C_VEL
LIN {X 0,Y 311.085,Z 569.956,A -85,B 0,C 180,E1 18160.824,E2 18160.824} C_VEL
LIN {X 0,Y 306.492,Z 558.753,A -85,B 0,C 180,E1 18167.159,E2 18167.159} C_VEL
LIN {X 0,Y 304.697,Z 554.03,A -85,B 0,C 180,E1 18171.055,E2 18171.055} C_VEL
LIN {X 0,Y 303.471,Z 550.747,A -85,B 0,C 180,E1 18178.572,E2 18178.572} C_VEL
LIN {X 0,Y 305.153,Z 555.454,A -85,B 0,C 180,E1 18186.048,E2 18186.048} C_VEL
LIN {X 0,Y 308.646,Z 564.753,A -85,B 0,C 180,E1 18192.259,E2 18192.259} C_VEL
LIN {X 0,Y 313.549,Z 578.642,A -85,B 0,C 180,E1 18198.293,E2 18198.293} C_VEL
LIN {X 0,Y 318.686,Z 597.798,A -85,B 0,C 180,E1 18204.188,E2 18204.188} C_VEL
LIN {X 0,Y 320.589,Z 611.201,A -85,B 0,C 180,E1 18207.379,E2 18207.379} C_VEL
LIN {X 0,Y 304.483,Z 649.808,A -85,B 0,C 180,E1 18210.929,E2 18210.929} C_VEL
LIN {X 0,Y 286.69,Z 684.931,A -85,B 0,C 180,E1 18215.78,E2 18215.78} C_VEL
LIN {X 0,Y 269.472,Z 714.876,A -85,B 0,C 180,E1 18221.883,E2 18221.883} C_VEL
LIN {X 0,Y 253.64,Z 740.371,A -85,B 0,C 180,E1 18229.464,E2 18229.464} C_VEL
LIN {X 0,Y 241.807,Z 760.485,A -85,B 0,C 180,E1 18238.366,E2 18238.366} C_VEL
LIN {X 0,Y 234.346,Z 775.332,A -85,B 0,C 180,E1 18248.333,E2 18248.333} C_VEL
LIN {X 0,Y 231.555,Z 783.117,A -85,B 0,C 180,E1 18256.77,E2 18256.77} C_VEL
LIN {X 0,Y 230.853,Z 787.48,A -85,B 0,C 180,E1 18266.239,E2 18266.239} C_VEL
LIN {X 0,Y 231.09,Z 787.878,A -85,B 0,C 180,E1 18270,E2 18270} C_VEL
LIN {X 0,Y 230.858,Z 786.329,A -85,B 0,C 180,E1 18277.537,E2 18277.537} C_VEL
LIN {X 0,Y 232.512,Z 780.075,A -85,B 0,C 180,E1 18287.04,E2 18287.04} C_VEL
LIN {X 0,Y 237.405,Z 768.544,A -85,B 0,C 180,E1 18296.769,E2 18296.769} C_VEL
LIN {X 0,Y 247.056,Z 751.287,A -85,B 0,C 180,E1 18306.149,E2 18306.149} C_VEL
LIN {X 0,Y 260.708,Z 729.324,A -85,B 0,C 180,E1 18314.182,E2 18314.182} C_VEL
LIN {X 0,Y 276.88,Z 702.572,A -85,B 0,C 180,E1 18320.917,E2 18320.917} C_VEL
LIN {X 0,Y 294.525,Z 670.428,A -85,B 0,C 180,E1 18326.462,E2 18326.462} C_VEL
LIN {X 0,Y 311.498,Z 634.289,A -85,B 0,C 180,E1 18330.681,E2 18330.681} C_VEL
LIN {X 0,Y 320.944,Z 609.982,A -85,B 0,C 180,E1 18332.778,E2 18332.778} C_VEL
LIN {X 0,Y 316.672,Z 589.336,A -85,B 0,C 180,E1 18338.251,E2 18338.251} C_VEL
LIN {X 0,Y 311.364,Z 571.794,A -85,B 0,C 180,E1 18344.481,E2 18344.481} C_VEL
LIN {X 0,Y 306.854,Z 559.812,A -85,B 0,C 180,E1 18350.791,E2 18350.791} C_VEL
LIN {X 0,Y 304.654,Z 553.848,A -85,B 0,C 180,E1 18355.724,E2 18355.724} C_VEL
LIN {X 0,Y 304.132,Z 553.158,A -85,B 0,C 180,E1 18357.11,E2 18357.11} C_VEL
LIN {X 0,Y 302.953,Z 554.364,A -85,B 0,C 180,E1 18359.561,E2 18359.561} C_VEL
LIN {X 0,Y 301.248,Z 559.392,A -85,B 0,C 180,E1 18363.648,E2 18363.648} C_VEL
LIN {X 0,Y 302.387,Z 561.635,A -85,B 0,C 180,E1 18368.637,E2 18368.637} C_VEL
LIN {X 0,Y 306.326,Z 572.64,A -85,B 0,C 180,E1 18376.508,E2 18376.508} C_VEL
LIN {X 0,Y 311.136,Z 587.383,A -85,B 0,C 180,E1 18382.907,E2 18382.907} C_VEL
LIN {X 0,Y 315.467,Z 606.035,A -85,B 0,C 180,E1 18388.678,E2 18388.678} C_VEL
LIN {X 0,Y 316.086,Z 612.302,A -85,B 0,C 180,E1 18390.194,E2 18390.194} C_VEL
LIN {X 0,Y 300.289,Z 647.892,A -85,B 0,C 180,E1 18393.512,E2 18393.512} C_VEL
LIN {X 0,Y 282.934,Z 679.78,A -85,B 0,C 180,E1 18397.992,E2 18397.992} C_VEL
LIN {X 0,Y 265.039,Z 707.79,A -85,B 0,C 180,E1 18403.842,E2 18403.842} C_VEL
LIN {X 0,Y 249.172,Z 730.359,A -85,B 0,C 180,E1 18410.916,E2 18410.916} C_VEL
LIN {X 0,Y 236.495,Z 747.889,A -85,B 0,C 180,E1 18419.19,E2 18419.19} C_VEL
LIN {X 0,Y 227.738,Z 761.291,A -85,B 0,C 180,E1 18429.296,E2 18429.296} C_VEL
LIN {X 0,Y 224.113,Z 768.195,A -85,B 0,C 180,E1 18438.306,E2 18438.306} C_VEL
LIN {X 0,Y 223.039,Z 771.018,A -85,B 0,C 180,E1 18446.107,E2 18446.107} C_VEL
LIN {X 0,Y 223.055,Z 770.989,A -85,B 0,C 180,E1 18453.892,E2 18453.892} C_VEL
LIN {X 0,Y 224.645,Z 766.984,A -85,B 0,C 180,E1 18463.645,E2 18463.645} C_VEL
LIN {X 0,Y 230.183,Z 757.205,A -85,B 0,C 180,E1 18474.275,E2 18474.275} C_VEL
LIN {X 0,Y 241.363,Z 741.034,A -85,B 0,C 180,E1 18484.374,E2 18484.374} C_VEL
LIN {X 0,Y 256.629,Z 719.797,A -85,B 0,C 180,E1 18492.656,E2 18492.656} C_VEL
LIN {X 0,Y 273.359,Z 695.138,A -85,B 0,C 180,E1 18498.996,E2 18498.996} C_VEL
LIN {X 0,Y 291.494,Z 664.617,A -85,B 0,C 180,E1 18504.255,E2 18504.255} C_VEL
LIN {X 0,Y 308.087,Z 631.174,A -85,B 0,C 180,E1 18508.112,E2 18508.112} C_VEL
LIN {X 0,Y 316.166,Z 610.851,A -85,B 0,C 180,E1 18509.944,E2 18509.944} C_VEL
LIN {X 0,Y 311.912,Z 590.626,A -85,B 0,C 180,E1 18515.837,E2 18515.837} C_VEL
LIN {X 0,Y 307.605,Z 576.486,A -85,B 0,C 180,E1 18521.368,E2 18521.368} C_VEL
LIN {X 0,Y 303.945,Z 566.507,A -85,B 0,C 180,E1 18527.049,E2 18527.049} C_VEL
LIN {X 0,Y 302.174,Z 561.424,A -85,B 0,C 180,E1 18531.357,E2 18531.357} C_VEL
LIN {X 0,Y 301.189,Z 558.535,A -85,B 0,C 180,E1 18537.12,E2 18537.12} C_VEL
LIN {X 0,Y 301.596,Z 560.557,A -85,B 0,C 180,E1 18542.879,E2 18542.879} C_VEL
LIN {X 0,Y 303.724,Z 566.458,A -85,B 0,C 180,E1 18548.602,E2 18548.602} C_VEL
LIN {X 0,Y 307.694,Z 578.054,A -85,B 0,C 180,E1 18554.972,E2 18554.972} C_VEL
LIN {X 0,Y 312.146,Z 594.279,A -85,B 0,C 180,E1 18560.92,E2 18560.92} C_VEL
LIN {X 0,Y 315.65,Z 613.411,A -85,B 0,C 180,E1 18566.221,E2 18566.221} C_VEL
LIN {X 0,Y 299.73,Z 650.656,A -85,B 0,C 180,E1 18569.743,E2 18569.743} C_VEL
LIN {X 0,Y 281.73,Z 684.908,A -85,B 0,C 180,E1 18574.479,E2 18574.479} C_VEL
LIN {X 0,Y 264.017,Z 714.532,A -85,B 0,C 180,E1 18580.546,E2 18580.546} C_VEL
LIN {X 0,Y 247.379,Z 740.161,A -85,B 0,C 180,E1 18588.269,E2 18588.269} C_VEL
LIN {X 0,Y 234.363,Z 760.877,A -85,B 0,C 180,E1 18597.719,E2 18597.719} C_VEL
LIN {X 0,Y 226.421,Z 775.806,A -85,B 0,C 180,E1 18608.315,E2 18608.315} C_VEL
LIN {X 0,Y 223.396,Z 784.109,A -85,B 0,C 180,E1 18618.268,E2 18618.268} C_VEL
LIN {X 0,Y 222.958,Z 787.192,A -85,B 0,C 180,E1 18626.106,E2 18626.106} C_VEL
LIN {X 0,Y 223.185,Z 787.59,A -85,B 0,C 180,E1 18630,E2 18630} C_VEL
LIN {X 0,Y 222.969,Z 786.039,A -85,B 0,C 180,E1 18637.806,E2 18637.806} C_VEL
LIN {X 0,Y 224.779,Z 779.78,A -85,B 0,C 180,E1 18647.645,E2 18647.645} C_VEL
LIN {X 0,Y 229.9,Z 768.585,A -85,B 0,C 180,E1 18657.453,E2 18657.453} C_VEL
LIN {X 0,Y 240.443,Z 750.97,A -85,B 0,C 180,E1 18667.309,E2 18667.309} C_VEL
LIN {X 0,Y 254.813,Z 728.991,A -85,B 0,C 180,E1 18675.484,E2 18675.484} C_VEL
LIN {X 0,Y 272.047,Z 701.722,A -85,B 0,C 180,E1 18682.365,E2 18682.365} C_VEL
LIN {X 0,Y 289.808,Z 670.502,A -85,B 0,C 180,E1 18687.751,E2 18687.751} C_VEL
LIN {X 0,Y 306.932,Z 635.354,A -85,B 0,C 180,E1 18691.86,E2 18691.86} C_VEL
LIN {X 0,Y 315.745,Z 613.469,A -85,B 0,C 180,E1 18693.787,E2 18693.787} C_VEL
LIN {X 0,Y 312.322,Z 594.614,A -85,B 0,C 180,E1 18699.009,E2 18699.009} C_VEL
LIN {X 0,Y 307.82,Z 578.193,A -85,B 0,C 180,E1 18705.034,E2 18705.034} C_VEL
LIN {X 0,Y 303.852,Z 566.692,A -85,B 0,C 180,E1 18711.402,E2 18711.402} C_VEL
LIN {X 0,Y 302.284,Z 561.409,A -85,B 0,C 180,E1 18715.69,E2 18715.69} C_VEL
LIN {X 0,Y 301.37,Z 559.219,A -85,B 0,C 180,E1 18719.998,E2 18719.998} C_VEL
LIN {X 0,Y 301.248,Z 559.392,A -85,B 0,C 180,E1 18723.648,E2 18723.648} C_VEL
LIN {X 0,Y 300.46,Z 564.501,A -85,B 0,C 180,E1 18726.821,E2 18726.821} C_VEL
LIN {X 0,Y 300.167,Z 570.79,A -85,B 0,C 180,E1 18729.972,E2 18729.972} C_VEL
LIN {X 0,Y 303.336,Z 580.607,A -85,B 0,C 180,E1 18736.656,E2 18736.656} C_VEL
LIN {X 0,Y 307.445,Z 594.672,A -85,B 0,C 180,E1 18742.786,E2 18742.786} C_VEL
LIN {X 0,Y 311.038,Z 614.081,A -85,B 0,C 180,E1 18748.808,E2 18748.808} C_VEL
LIN {X 0,Y 310.622,Z 616.646,A -85,B 0,C 180,E1 18749.237,E2 18749.237} C_VEL
LIN {X 0,Y 294.332,Z 651.466,A -85,B 0,C 180,E1 18752.596,E2 18752.596} C_VEL
LIN {X 0,Y 276.21,Z 683.095,A -85,B 0,C 180,E1 18757.202,E2 18757.202} C_VEL
LIN {X 0,Y 258.324,Z 709.814,A -85,B 0,C 180,E1 18763.009,E2 18763.009} C_VEL
LIN {X 0,Y 242.128,Z 731.72,A -85,B 0,C 180,E1 18770.135,E2 18770.135} C_VEL
LIN {X 0,Y 228.368,Z 749.765,A -85,B 0,C 180,E1 18779.157,E2 18779.157} C_VEL
LIN {X 0,Y 220.217,Z 761.584,A -85,B 0,C 180,E1 18788.555,E2 18788.555} C_VEL
LIN {X 0,Y 216.057,Z 768.999,A -85,B 0,C 180,E1 18798.803,E2 18798.803} C_VEL
LIN {X 0,Y 215.322,Z 771.644,A -85,B 0,C 180,E1 18810,E2 18810} C_VEL
LIN {X 0,Y 216.098,Z 768.91,A -85,B 0,C 180,E1 18821.252,E2 18821.252} C_VEL
LIN {X 0,Y 220.285,Z 761.438,A -85,B 0,C 180,E1 18831.485,E2 18831.485} C_VEL
LIN {X 0,Y 229.738,Z 748.018,A -85,B 0,C 180,E1 18841.82,E2 18841.82} C_VEL
LIN {X 0,Y 244.694,Z 728.282,A -85,B 0,C 180,E1 18851.107,E2 18851.107} C_VEL
LIN {X 0,Y 262.749,Z 703.374,A -85,B 0,C 180,E1 18858.517,E2 18858.517} C_VEL
LIN {X 0,Y 281.382,Z 674.457,A -85,B 0,C 180,E1 18864.147,E2 18864.147} C_VEL
LIN {X 0,Y 298.917,Z 642.325,A -85,B 0,C 180,E1 18868.307,E2 18868.307} C_VEL
LIN {X 0,Y 311.043,Z 614.804,A -85,B 0,C 180,E1 18870.876,E2 18870.876} C_VEL
LIN {X 0,Y 307.521,Z 595.5,A -85,B 0,C 180,E1 18876.808,E2 18876.808} C_VEL
LIN {X 0,Y 303.625,Z 581.715,A -85,B 0,C 180,E1 18882.594,E2 18882.594} C_VEL
LIN {X 0,Y 300.583,Z 572.417,A -85,B 0,C 180,E1 18888.379,E2 18888.379} C_VEL
LIN {X 0,Y 299.63,Z 569.054,A -85,B 0,C 180,E1 18891.283,E2 18891.283} C_VEL
LIN {X 0,Y 298.654,Z 566.047,A -85,B 0,C 180,E1 18897.096,E2 18897.096} C_VEL
LIN {X 0,Y 299.056,Z 568.072,A -85,B 0,C 180,E1 18902.903,E2 18902.903} C_VEL
LIN {X 0,Y 301.326,Z 575.182,A -85,B 0,C 180,E1 18909.4,E2 18909.4} C_VEL
LIN {X 0,Y 305.013,Z 587.784,A -85,B 0,C 180,E1 18915.844,E2 18915.844} C_VEL
LIN {X 0,Y 308.91,Z 605.638,A -85,B 0,C 180,E1 18922.062,E2 18922.062} C_VEL
LIN {X 0,Y 310.258,Z 618.052,A -85,B 0,C 180,E1 18925.366,E2 18925.366} C_VEL
LIN {X 0,Y 293.796,Z 654.082,A -85,B 0,C 180,E1 18928.821,E2 18928.821} C_VEL
LIN {X 0,Y 276.131,Z 686.215,A -85,B 0,C 180,E1 18933.367,E2 18933.367} C_VEL
LIN {X 0,Y 257.701,Z 715.69,A -85,B 0,C 180,E1 18939.541,E2 18939.541} C_VEL
LIN {X 0,Y 240.461,Z 740.964,A -85,B 0,C 180,E1 18947.398,E2 18947.398} C_VEL
LIN {X 0,Y 227.409,Z 760.567,A -85,B 0,C 180,E1 18956.605,E2 18956.605} C_VEL
LIN {X 0,Y 218.794,Z 775.609,A -85,B 0,C 180,E1 18967.628,E2 18967.628} C_VEL
LIN {X 0,Y 215.566,Z 783.816,A -85,B 0,C 180,E1 18977.835,E2 18977.835} C_VEL
LIN {X 0,Y 215.04,Z 786.903,A -85,B 0,C 180,E1 18985.962,E2 18985.962} C_VEL
LIN {X 0,Y 215.28,Z 787.303,A -85,B 0,C 180,E1 18990,E2 18990} C_VEL
LIN {X 0,Y 215.168,Z 784.932,A -85,B 0,C 180,E1 18999.904,E2 18999.904} C_VEL
LIN {X 0,Y 217.071,Z 779.484,A -85,B 0,C 180,E1 19008.294,E2 19008.294} C_VEL
LIN {X 0,Y 222.632,Z 768.281,A -85,B 0,C 180,E1 19018.429,E2 19018.429} C_VEL
LIN {X 0,Y 232.955,Z 752.11,A -85,B 0,C 180,E1 19027.872,E2 19027.872} C_VEL
LIN {X 0,Y 248.058,Z 730.193,A -85,B 0,C 180,E1 19036.377,E2 19036.377} C_VEL
LIN {X 0,Y 266.428,Z 702.449,A -85,B 0,C 180,E1 19043.545,E2 19043.545} C_VEL
LIN {X 0,Y 285.286,Z 670.566,A -85,B 0,C 180,E1 19049.072,E2 19049.072} C_VEL
LIN {X 0,Y 303.346,Z 634.511,A -85,B 0,C 180,E1 19053.242,E2 19053.242} C_VEL
LIN {X 0,Y 310.337,Z 618.101,A -85,B 0,C 180,E1 19054.652,E2 19054.652} C_VEL
LIN {X 0,Y 308.481,Z 602.811,A -85,B 0,C 180,E1 19058.842,E2 19058.842} C_VEL
LIN {X 0,Y 304.733,Z 586.182,A -85,B 0,C 180,E1 19064.879,E2 19064.879} C_VEL
LIN {X 0,Y 301.115,Z 574.378,A -85,B 0,C 180,E1 19071.323,E2 19071.323} C_VEL
LIN {X 0,Y 299.248,Z 568.202,A -85,B 0,C 180,E1 19077.098,E2 19077.098} C_VEL
LIN {X 0,Y 298.737,Z 566.572,A -85,B 0,C 180,E1 19082.903,E2 19082.903} C_VEL
LIN {X 0,Y 300.167,Z 570.79,A -85,B 0,C 180,E1 19089.972,E2 19089.972} C_VEL
LIN {X 0,Y 300.131,Z 575.979,A -85,B 0,C 180,E1 19092.274,E2 19092.274} C_VEL
LIN {X 0,Y 299.766,Z 586.844,A -85,B 0,C 180,E1 19095.968,E2 19095.968} C_VEL
LIN {X 0,Y 303.139,Z 600.105,A -85,B 0,C 180,E1 19101.996,E2 19101.996} C_VEL
LIN {X 0,Y 306.03,Z 618.147,A -85,B 0,C 180,E1 19107.87,E2 19107.87} C_VEL
LIN {X 0,Y 300.218,Z 632.069,A -85,B 0,C 180,E1 19109.216,E2 19109.216} C_VEL
LIN {X 0,Y 282.376,Z 665.884,A -85,B 0,C 180,E1 19113.088,E2 19113.088} C_VEL
LIN {X 0,Y 262.962,Z 696.197,A -85,B 0,C 180,E1 19118.323,E2 19118.323} C_VEL
LIN {X 0,Y 243.982,Z 721.975,A -85,B 0,C 180,E1 19125.17,E2 19125.17} C_VEL
LIN {X 0,Y 228.078,Z 741.855,A -85,B 0,C 180,E1 19133.31,E2 19133.31} C_VEL
LIN {X 0,Y 215.557,Z 757.922,A -85,B 0,C 180,E1 19143.959,E2 19143.959} C_VEL
LIN {X 0,Y 209.139,Z 767.632,A -85,B 0,C 180,E1 19155.322,E2 19155.322} C_VEL
LIN {X 0,Y 207.251,Z 771.594,A -85,B 0,C 180,E1 19165.81,E2 19165.81} C_VEL
LIN {X 0,Y 207.431,Z 771.931,A -85,B 0,C 180,E1 19170,E2 19170} C_VEL
LIN {X 0,Y 207.59,Z 770.494,A -85,B 0,C 180,E1 19178.388,E2 19178.388} C_VEL
LIN {X 0,Y 210.844,Z 764.717,A -85,B 0,C 180,E1 19188.854,E2 19188.854} C_VEL
LIN {X 0,Y 219.645,Z 752.497,A -85,B 0,C 180,E1 19200.175,E2 19200.175} C_VEL
LIN {X 0,Y 233.187,Z 735.504,A -85,B 0,C 180,E1 19209.568,E2 19209.568} C_VEL
LIN {X 0,Y 250.909,Z 712.733,A -85,B 0,C 180,E1 19217.518,E2 19217.518} C_VEL
LIN {X 0,Y 270.658,Z 684.516,A -85,B 0,C 180,E1 19223.846,E2 19223.846} C_VEL
LIN {X 0,Y 289.393,Z 653.11,A -85,B 0,C 180,E1 19228.458,E2 19228.458} C_VEL
LIN {X 0,Y 305.969,Z 618.409,A -85,B 0,C 180,E1 19231.934,E2 19231.934} C_VEL
LIN {X 0,Y 303.359,Z 601.801,A -85,B 0,C 180,E1 19237.248,E2 19237.248} C_VEL
LIN {X 0,Y 299.999,Z 588.041,A -85,B 0,C 180,E1 19243.208,E2 19243.208} C_VEL
LIN {X 0,Y 297.288,Z 578.522,A -85,B 0,C 180,E1 19249.456,E2 19249.456} C_VEL
LIN {X 0,Y 296.067,Z 574.961,A -85,B 0,C 180,E1 19254.132,E2 19254.132} C_VEL
LIN {X 0,Y 295.999,Z 573.54,A -85,B 0,C 180,E1 19257.07,E2 19257.07} C_VEL
LIN {X 0,Y 296.32,Z 575.504,A -85,B 0,C 180,E1 19262.93,E2 19262.93} C_VEL
LIN {X 0,Y 298.358,Z 582.897,A -85,B 0,C 180,E1 19269.494,E2 19269.494} C_VEL
LIN {X 0,Y 301.487,Z 595.387,A -85,B 0,C 180,E1 19275.851,E2 19275.851} C_VEL
LIN {X 0,Y 304.581,Z 612.596,A -85,B 0,C 180,E1 19281.875,E2 19281.875} C_VEL
LIN {X 0,Y 305.418,Z 620.464,A -85,B 0,C 180,E1 19284.141,E2 19284.141} C_VEL
LIN {X 0,Y 288.461,Z 656.488,A -85,B 0,C 180,E1 19287.738,E2 19287.738} C_VEL
LIN {X 0,Y 269.492,Z 689.467,A -85,B 0,C 180,E1 19292.566,E2 19292.566} C_VEL
LIN {X 0,Y 250.61,Z 718.076,A -85,B 0,C 180,E1 19298.808,E2 19298.808} C_VEL
LIN {X 0,Y 233.612,Z 741.767,A -85,B 0,C 180,E1 19306.476,E2 19306.476} C_VEL
LIN {X 0,Y 220.519,Z 760.338,A -85,B 0,C 180,E1 19315.476,E2 19315.476} C_VEL
LIN {X 0,Y 211.246,Z 775.309,A -85,B 0,C 180,E1 19326.783,E2 19326.783} C_VEL
LIN {X 0,Y 207.722,Z 783.522,A -85,B 0,C 180,E1 19337.369,E2 19337.369} C_VEL
LIN {X 0,Y 207.147,Z 786.615,A -85,B 0,C 180,E1 19345.808,E2 19345.808} C_VEL
LIN {X 0,Y 207.39,Z 787.016,A -85,B 0,C 180,E1 19350,E2 19350} C_VEL
LIN {X 0,Y 207.187,Z 785.458,A -85,B 0,C 180,E1 19358.404,E2 19358.404} C_VEL
LIN {X 0,Y 209.267,Z 779.487,A -85,B 0,C 180,E1 19368.608,E2 19368.608} C_VEL
LIN {X 0,Y 215.437,Z 767.976,A -85,B 0,C 180,E1 19379.47,E2 19379.47} C_VEL
LIN {X 0,Y 226.309,Z 752.076,A -85,B 0,C 180,E1 19389.022,E2 19389.022} C_VEL
LIN {X 0,Y 242.646,Z 729.547,A -85,B 0,C 180,E1 19397.889,E2 19397.889} C_VEL
LIN {X 0,Y 261.363,Z 702.49,A -85,B 0,C 180,E1 19404.914,E2 19404.914} C_VEL
LIN {X 0,Y 280.872,Z 670.69,A -85,B 0,C 180,E1 19410.432,E2 19410.432} C_VEL
LIN {X 0,Y 299.18,Z 635.357,A -85,B 0,C 180,E1 19414.508,E2 19414.508} C_VEL
LIN {X 0,Y 305.546,Z 620.483,A -85,B 0,C 180,E1 19415.87,E2 19415.87} C_VEL
LIN {X 0,Y 303.039,Z 602.595,A -85,B 0,C 180,E1 19421.431,E2 19421.431} C_VEL
LIN {X 0,Y 299.875,Z 588.558,A -85,B 0,C 180,E1 19427.384,E2 19427.384} C_VEL
LIN {X 0,Y 297.541,Z 580.226,A -85,B 0,C 180,E1 19432.69,E2 19432.69} C_VEL
LIN {X 0,Y 296.5,Z 575.647,A -85,B 0,C 180,E1 19437.072,E2 19437.072} C_VEL
LIN {X 0,Y 296.068,Z 574.032,A -85,B 0,C 180,E1 19442.929,E2 19442.929} C_VEL
LIN {X 0,Y 297.171,Z 577.942,A -85,B 0,C 180,E1 19449.679,E2 19449.679} C_VEL
LIN {X 0,Y 299.766,Z 586.844,A -85,B 0,C 180,E1 19455.968,E2 19455.968} C_VEL
LIN {X 0,Y 299.845,Z 593.443,A -85,B 0,C 180,E1 19458.14,E2 19458.14} C_VEL
LIN {X 0,Y 299,Z 606.456,A -85,B 0,C 180,E1 19461.58,E2 19461.58} C_VEL
LIN {X 0,Y 301.071,Z 622.228,A -85,B 0,C 180,E1 19466.907,E2 19466.907} C_VEL
LIN {X 0,Y 283.198,Z 657.526,A -85,B 0,C 180,E1 19470.547,E2 19470.547} C_VEL
LIN {X 0,Y 263.81,Z 688.333,A -85,B 0,C 180,E1 19475.284,E2 19475.284} C_VEL
LIN {X 0,Y 243.557,Z 715.708,A -85,B 0,C 180,E1 19481.754,E2 19481.754} C_VEL
LIN {X 0,Y 225.794,Z 737.274,A -85,B 0,C 180,E1 19489.69,E2 19489.69} C_VEL
LIN {X 0,Y 211.314,Z 754.475,A -85,B 0,C 180,E1 19499.896,E2 19499.896} C_VEL
LIN {X 0,Y 203.259,Z 765.091,A -85,B 0,C 180,E1 19510.414,E2 19510.414} C_VEL
LIN {X 0,Y 199.721,Z 770.831,A -85,B 0,C 180,E1 19521.279,E2 19521.279} C_VEL
LIN {X 0,Y 199.528,Z 772.218,A -85,B 0,C 180,E1 19530,E2 19530} C_VEL
LIN {X 0,Y 199.972,Z 770.231,A -85,B 0,C 180,E1 19540.211,E2 19540.211} C_VEL
LIN {X 0,Y 203.277,Z 765.008,A -85,B 0,C 180,E1 19549.584,E2 19549.584} C_VEL
LIN {X 0,Y 212.847,Z 752.601,A -85,B 0,C 180,E1 19561.405,E2 19561.405} C_VEL
LIN {X 0,Y 228.32,Z 734.215,A -85,B 0,C 180,E1 19571.542,E2 19571.542} C_VEL
LIN {X 0,Y 246.151,Z 712.242,A -85,B 0,C 180,E1 19579.13,E2 19579.13} C_VEL
LIN {X 0,Y 265.547,Z 685.585,A -85,B 0,C 180,E1 19585.115,E2 19585.115} C_VEL
LIN {X 0,Y 284.66,Z 654.748,A -85,B 0,C 180,E1 19589.676,E2 19589.676} C_VEL
LIN {X 0,Y 300.924,Z 621.906,A -85,B 0,C 180,E1 19593.079,E2 19593.079} C_VEL
LIN {X 0,Y 298.448,Z 604.144,A -85,B 0,C 180,E1 19599.203,E2 19599.203} C_VEL
LIN {X 0,Y 295.728,Z 591.944,A -85,B 0,C 180,E1 19605.171,E2 19605.171} C_VEL
LIN {X 0,Y 293.91,Z 584.189,A -85,B 0,C 180,E1 19611.112,E2 19611.112} C_VEL
LIN {X 0,Y 293.124,Z 580.935,A -85,B 0,C 180,E1 19617.041,E2 19617.041} C_VEL
LIN {X 0,Y 293.442,Z 582.898,A -85,B 0,C 180,E1 19622.959,E2 19622.959} C_VEL
LIN {X 0,Y 295.109,Z 590.54,A -85,B 0,C 180,E1 19629.599,E2 19629.599} C_VEL
LIN {X 0,Y 297.533,Z 601.809,A -85,B 0,C 180,E1 19635.403,E2 19635.403} C_VEL
LIN {X 0,Y 299.9,Z 618.472,A -85,B 0,C 180,E1 19641.393,E2 19641.393} C_VEL
LIN {X 0,Y 300.149,Z 625.177,A -85,B 0,C 180,E1 19643.248,E2 19643.248} C_VEL
LIN {X 0,Y 281.908,Z 661.397,A -85,B 0,C 180,E1 19646.943,E2 19646.943} C_VEL
LIN {X 0,Y 261.439,Z 694.816,A -85,B 0,C 180,E1 19652.111,E2 19652.111} C_VEL
LIN {X 0,Y 241.293,Z 723.435,A -85,B 0,C 180,E1 19658.863,E2 19658.863} C_VEL
LIN {X 0,Y 223.591,Z 746.938,A -85,B 0,C 180,E1 19667.375,E2 19667.375} C_VEL
LIN {X 0,Y 210.378,Z 764.833,A -85,B 0,C 180,E1 19677.331,E2 19677.331} C_VEL
LIN {X 0,Y 202.217,Z 778.022,A -85,B 0,C 180,E1 19689.142,E2 19689.142} C_VEL
LIN {X 0,Y 199.898,Z 783.228,A -85,B 0,C 180,E1 19696.865,E2 19696.865} C_VEL
LIN {X 0,Y 199.227,Z 786.325,A -85,B 0,C 180,E1 19705.641,E2 19705.641} C_VEL
LIN {X 0,Y 199.484,Z 786.728,A -85,B 0,C 180,E1 19710,E2 19710} C_VEL
LIN {X 0,Y 199.31,Z 785.033,A -85,B 0,C 180,E1 19719.062,E2 19719.062} C_VEL
LIN {X 0,Y 201.536,Z 779.32,A -85,B 0,C 180,E1 19729.174,E2 19729.174} C_VEL
LIN {X 0,Y 208.324,Z 767.674,A -85,B 0,C 180,E1 19740.582,E2 19740.582} C_VEL
LIN {X 0,Y 221.222,Z 750.096,A -85,B 0,C 180,E1 19751.164,E2 19751.164} C_VEL
LIN {X 0,Y 237.98,Z 727.992,A -85,B 0,C 180,E1 19759.773,E2 19759.773} C_VEL
LIN {X 0,Y 257.879,Z 700.337,A -85,B 0,C 180,E1 19766.792,E2 19766.792} C_VEL
LIN {X 0,Y 277.87,Z 668.628,A -85,B 0,C 180,E1 19772.126,E2 19772.126} C_VEL
LIN {X 0,Y 295.995,Z 634.386,A -85,B 0,C 180,E1 19775.971,E2 19775.971} C_VEL
LIN {X 0,Y 300.504,Z 624.071,A -85,B 0,C 180,E1 19776.98,E2 19776.98} C_VEL
LIN {X 0,Y 298.54,Z 607.221,A -85,B 0,C 180,E1 19782.497,E2 19782.497} C_VEL
LIN {X 0,Y 296.085,Z 594.511,A -85,B 0,C 180,E1 19788.196,E2 19788.196} C_VEL
LIN {X 0,Y 293.99,Z 584.807,A -85,B 0,C 180,E1 19795.032,E2 19795.032} C_VEL
LIN {X 0,Y 293.28,Z 581.561,A -85,B 0,C 180,E1 19799.998,E2 19799.998} C_VEL
LIN {X 0,Y 293.343,Z 582.703,A -85,B 0,C 180,E1 19805.923,E2 19805.923} C_VEL
LIN {X 0,Y 294.431,Z 586.705,A -85,B 0,C 180,E1 19810.792,E2 19810.792} C_VEL
LIN {X 0,Y 296.99,Z 596.669,A -85,B 0,C 180,E1 19817.227,E2 19817.227} C_VEL
LIN {X 0,Y 299,Z 606.456,A -85,B 0,C 180,E1 19821.58,E2 19821.58} C_VEL
LIN {X 0,Y 298.245,Z 612.216,A -85,B 0,C 180,E1 19822.848,E2 19822.848} C_VEL
LIN {X 0,Y 295.799,Z 622.114,A -85,B 0,C 180,E1 19824.561,E2 19824.561} C_VEL
LIN {X 0,Y 295.779,Z 622.927,A -85,B 0,C 180,E1 19824.803,E2 19824.803} C_VEL
LIN {X 0,Y 295.673,Z 627.042,A -85,B 0,C 180,E1 19825.998,E2 19825.998} C_VEL
LIN {X 0,Y 278.032,Z 659.87,A -85,B 0,C 180,E1 19829.385,E2 19829.385} C_VEL
LIN {X 0,Y 258.142,Z 690.203,A -85,B 0,C 180,E1 19834.137,E2 19834.137} C_VEL
LIN {X 0,Y 238.274,Z 716.023,A -85,B 0,C 180,E1 19840.31,E2 19840.31} C_VEL
LIN {X 0,Y 219.279,Z 738.025,A -85,B 0,C 180,E1 19848.546,E2 19848.546} C_VEL
LIN {X 0,Y 204.346,Z 754.771,A -85,B 0,C 180,E1 19858.757,E2 19858.757} C_VEL
LIN {X 0,Y 195.7,Z 765.383,A -85,B 0,C 180,E1 19869.625,E2 19869.625} C_VEL
LIN {X 0,Y 191.87,Z 771.12,A -85,B 0,C 180,E1 19880.919,E2 19880.919} C_VEL
LIN {X 0,Y 191.639,Z 772.505,A -85,B 0,C 180,E1 19890,E2 19890} C_VEL
LIN {X 0,Y 191.901,Z 771.072,A -85,B 0,C 180,E1 19899.08,E2 19899.08} C_VEL
LIN {X 0,Y 195.72,Z 765.301,A -85,B 0,C 180,E1 19910.373,E2 19910.373} C_VEL
LIN {X 0,Y 205.998,Z 752.902,A -85,B 0,C 180,E1 19922.576,E2 19922.576} C_VEL
LIN {X 0,Y 222.327,Z 734.527,A -85,B 0,C 180,E1 19932.925,E2 19932.925} C_VEL
LIN {X 0,Y 241.279,Z 712.122,A -85,B 0,C 180,E1 19940.709,E2 19940.709} C_VEL
LIN {X 0,Y 262.191,Z 684.276,A -85,B 0,C 180,E1 19946.846,E2 19946.846} C_VEL
LIN {X 0,Y 281.666,Z 653.494,A -85,B 0,C 180,E1 19951.268,E2 19951.268} C_VEL
LIN {X 0,Y 295.494,Z 626.959,A -85,B 0,C 180,E1 19953.934,E2 19953.934} C_VEL
LIN {X 0,Y 294.993,Z 615.881,A -85,B 0,C 180,E1 19957.504,E2 19957.504} C_VEL
LIN {X 0,Y 292.827,Z 602.301,A -85,B 0,C 180,E1 19963.481,E2 19963.481} C_VEL
LIN {X 0,Y 291.038,Z 593.606,A -85,B 0,C 180,E1 19969.227,E2 19969.227} C_VEL
LIN {X 0,Y 290.08,Z 589.703,A -85,B 0,C 180,E1 19974.01,E2 19974.01} C_VEL
LIN {X 0,Y 290.073,Z 588.259,A -85,B 0,C 180,E1 19977.01,E2 19977.01} C_VEL
LIN {X 0,Y 290.294,Z 590.215,A -85,B 0,C 180,E1 19982.991,E2 19982.991} C_VEL
LIN {X 0,Y 291.737,Z 597.884,A -85,B 0,C 180,E1 19989.559,E2 19989.559} C_VEL
LIN {X 0,Y 293.801,Z 609.884,A -85,B 0,C 180,E1 19995.698,E2 19995.698} C_VEL
LIN {X 0,Y 295.371,Z 627.686,A -85,B 0,C 180,E1 20001.965,E2 20001.965} C_VEL
LIN {X 0,Y 277.445,Z 662.408,A -85,B 0,C 180,E1 20005.622,E2 20005.622} C_VEL
LIN {X 0,Y 257.176,Z 694.458,A -85,B 0,C 180,E1 20010.565,E2 20010.565} C_VEL
LIN {X 0,Y 236.241,Z 723.107,A -85,B 0,C 180,E1 20017.317,E2 20017.317} C_VEL
LIN {X 0,Y 217.492,Z 746.619,A -85,B 0,C 180,E1 20025.879,E2 20025.879} C_VEL
LIN {X 0,Y 203.404,Z 764.608,A -85,B 0,C 180,E1 20036.135,E2 20036.135} C_VEL
LIN {X 0,Y 195.156,Z 776.744,A -85,B 0,C 180,E1 20047.174,E2 20047.174} C_VEL
LIN {X 0,Y 192.075,Z 782.934,A -85,B 0,C 180,E1 20056.32,E2 20056.32} C_VEL
LIN {X 0,Y 191.312,Z 786.036,A -85,B 0,C 180,E1 20065.46,E2 20065.46} C_VEL
LIN {X 0,Y 191.595,Z 786.441,A -85,B 0,C 180,E1 20070,E2 20070} C_VEL
LIN {X 0,Y 191.435,Z 784.878,A -85,B 0,C 180,E1 20079.102,E2 20079.102} C_VEL
LIN {X 0,Y 194.158,Z 778.523,A -85,B 0,C 180,E1 20090.651,E2 20090.651} C_VEL
LIN {X 0,Y 201.274,Z 767.369,A -85,B 0,C 180,E1 20101.775,E2 20101.775} C_VEL
LIN {X 0,Y 215.068,Z 749.784,A -85,B 0,C 180,E1 20112.613,E2 20112.613} C_VEL
LIN {X 0,Y 232.681,Z 727.661,A -85,B 0,C 180,E1 20121.341,E2 20121.341} C_VEL
LIN {X 0,Y 253.448,Z 699.979,A -85,B 0,C 180,E1 20128.355,E2 20128.355} C_VEL
LIN {X 0,Y 274.206,Z 668.091,A -85,B 0,C 180,E1 20133.66,E2 20133.66} C_VEL
LIN {X 0,Y 293.03,Z 633.378,A -85,B 0,C 180,E1 20137.467,E2 20137.467} C_VEL
LIN {X 0,Y 295.465,Z 627.794,A -85,B 0,C 180,E1 20138.04,E2 20138.04} C_VEL
LIN {X 0,Y 294.131,Z 611.913,A -85,B 0,C 180,E1 20143.553,E2 20143.553} C_VEL
LIN {X 0,Y 292.293,Z 600.661,A -85,B 0,C 180,E1 20148.874,E2 20148.874} C_VEL
LIN {X 0,Y 290.564,Z 591.253,A -85,B 0,C 180,E1 20155.993,E2 20155.993} C_VEL
LIN {X 0,Y 290.21,Z 588.843,A -85,B 0,C 180,E1 20159.998,E2 20159.998} C_VEL
LIN {X 0,Y 290.21,Z 590.025,A -85,B 0,C 180,E1 20165.987,E2 20165.987} C_VEL
LIN {X 0,Y 291.186,Z 594.18,A -85,B 0,C 180,E1 20170.913,E2 20170.913} C_VEL
LIN {X 0,Y 293.277,Z 604.029,A -85,B 0,C 180,E1 20177.265,E2 20177.265} C_VEL
LIN {X 0,Y 295.448,Z 618.667,A -85,B 0,C 180,E1 20183.385,E2 20183.385} C_VEL
LIN {X 0,Y 295.779,Z 622.927,A -85,B 0,C 180,E1 20184.803,E2 20184.803} C_VEL
LIN {X 0,Y 293.745,Z 628.38,A -85,B 0,C 180,E1 20185.525,E2 20185.525} C_VEL
LIN {X 0,Y 284.363,Z 642.815,A -85,B 0,C 180,E1 20185.986,E2 20185.986} C_VEL
LIN {X 0,Y 264.457,Z 675.495,A -85,B 0,C 180,E1 20190.068,E2 20190.068} C_VEL
LIN {X 0,Y 243.807,Z 703.476,A -85,B 0,C 180,E1 20195.402,E2 20195.402} C_VEL
LIN {X 0,Y 222.948,Z 727.882,A -85,B 0,C 180,E1 20202.659,E2 20202.659} C_VEL
LIN {X 0,Y 204.289,Z 747.879,A -85,B 0,C 180,E1 20212.358,E2 20212.358} C_VEL
LIN {X 0,Y 191.219,Z 762.081,A -85,B 0,C 180,E1 20224.182,E2 20224.182} C_VEL
LIN {X 0,Y 185.248,Z 769.645,A -85,B 0,C 180,E1 20235.806,E2 20235.806} C_VEL
LIN {X 0,Y 183.552,Z 772.458,A -85,B 0,C 180,E1 20245.268,E2 20245.268} C_VEL
LIN {X 0,Y 183.735,Z 772.792,A -85,B 0,C 180,E1 20250,E2 20250} C_VEL
LIN {X 0,Y 184.077,Z 771.362,A -85,B 0,C 180,E1 20259.469,E2 20259.469} C_VEL
LIN {X 0,Y 188.208,Z 765.618,A -85,B 0,C 180,E1 20271.182,E2 20271.182} C_VEL
LIN {X 0,Y 198.714,Z 753.769,A -85,B 0,C 180,E1 20283.402,E2 20283.402} C_VEL
LIN {X 0,Y 215.538,Z 735.893,A -85,B 0,C 180,E1 20293.925,E2 20293.925} C_VEL
LIN {X 0,Y 235.78,Z 713.043,A -85,B 0,C 180,E1 20302.06,E2 20302.06} C_VEL
LIN {X 0,Y 256.826,Z 686.181,A -85,B 0,C 180,E1 20308.066,E2 20308.066} C_VEL
LIN {X 0,Y 277.221,Z 655.15,A -85,B 0,C 180,E1 20312.567,E2 20312.567} C_VEL
LIN {X 0,Y 290.355,Z 631.07,A -85,B 0,C 180,E1 20315.01,E2 20315.01} C_VEL
LIN {X 0,Y 290.524,Z 622.214,A -85,B 0,C 180,E1 20317.875,E2 20317.875} C_VEL
LIN {X 0,Y 288.874,Z 608.469,A -85,B 0,C 180,E1 20324.101,E2 20324.101} C_VEL
LIN {X 0,Y 287.344,Z 599.036,A -85,B 0,C 180,E1 20330.907,E2 20330.907} C_VEL
LIN {X 0,Y 286.865,Z 595.522,A -85,B 0,C 180,E1 20336.976,E2 20336.976} C_VEL
LIN {X 0,Y 287.061,Z 597.515,A -85,B 0,C 180,E1 20343.025,E2 20343.025} C_VEL
LIN {X 0,Y 288.086,Z 605.336,A -85,B 0,C 180,E1 20349.681,E2 20349.681} C_VEL
LIN {X 0,Y 289.494,Z 615.905,A -85,B 0,C 180,E1 20355.16,E2 20355.16} C_VEL
LIN {X 0,Y 290.408,Z 631.639,A -85,B 0,C 180,E1 20360.931,E2 20360.931} C_VEL
LIN {X 0,Y 271.839,Z 665.589,A -85,B 0,C 180,E1 20364.546,E2 20364.546} C_VEL
LIN {X 0,Y 250.998,Z 696.93,A -85,B 0,C 180,E1 20369.503,E2 20369.503} C_VEL
LIN {X 0,Y 230.439,Z 723.853,A -85,B 0,C 180,E1 20376.016,E2 20376.016} C_VEL
LIN {X 0,Y 211.601,Z 746.303,A -85,B 0,C 180,E1 20384.311,E2 20384.311} C_VEL
LIN {X 0,Y 196.432,Z 764.484,A -85,B 0,C 180,E1 20394.934,E2 20394.934} C_VEL
LIN {X 0,Y 187.637,Z 776.443,A -85,B 0,C 180,E1 20406.204,E2 20406.204} C_VEL
LIN {X 0,Y 184.282,Z 782.641,A -85,B 0,C 180,E1 20415.73,E2 20415.73} C_VEL
LIN {X 0,Y 183.393,Z 785.747,A -85,B 0,C 180,E1 20425.264,E2 20425.264} C_VEL
LIN {X 0,Y 183.686,Z 786.154,A -85,B 0,C 180,E1 20430,E2 20430} C_VEL
LIN {X 0,Y 183.567,Z 784.588,A -85,B 0,C 180,E1 20439.495,E2 20439.495} C_VEL
LIN {X 0,Y 186.548,Z 778.227,A -85,B 0,C 180,E1 20451.535,E2 20451.535} C_VEL
LIN {X 0,Y 195.381,Z 765.793,A -85,B 0,C 180,E1 20464.065,E2 20464.065} C_VEL
LIN {X 0,Y 210.388,Z 747.839,A -85,B 0,C 180,E1 20474.961,E2 20474.961} C_VEL
LIN {X 0,Y 229.158,Z 725.502,A -85,B 0,C 180,E1 20483.514,E2 20483.514} C_VEL
LIN {X 0,Y 250.016,Z 698.528,A -85,B 0,C 180,E1 20490.185,E2 20490.185} C_VEL
LIN {X 0,Y 270.679,Z 667.689,A -85,B 0,C 180,E1 20495.211,E2 20495.211} C_VEL
LIN {X 0,Y 289.468,Z 634.023,A -85,B 0,C 180,E1 20498.852,E2 20498.852} C_VEL
LIN {X 0,Y 290.49,Z 630.728,A -85,B 0,C 180,E1 20499.401,E2 20499.401} C_VEL
LIN {X 0,Y 289.567,Z 616.108,A -85,B 0,C 180,E1 20504.844,E2 20504.844} C_VEL
LIN {X 0,Y 288.212,Z 605.808,A -85,B 0,C 180,E1 20510.171,E2 20510.171} C_VEL
LIN {X 0,Y 287.204,Z 597.709,A -85,B 0,C 180,E1 20516.977,E2 20516.977} C_VEL
LIN {X 0,Y 286.998,Z 596.102,A -85,B 0,C 180,E1 20519.998,E2 20519.998} C_VEL
LIN {X 0,Y 287.004,Z 597.299,A -85,B 0,C 180,E1 20526.054,E2 20526.054} C_VEL
LIN {X 0,Y 287.667,Z 601.053,A -85,B 0,C 180,E1 20530.613,E2 20530.613} C_VEL
LIN {X 0,Y 289.466,Z 611.82,A -85,B 0,C 180,E1 20537.501,E2 20537.501} C_VEL
LIN {X 0,Y 290.839,Z 625.89,A -85,B 0,C 180,E1 20543.366,E2 20543.366} C_VEL
LIN {X 0,Y 290.383,Z 631.408,A -85,B 0,C 180,E1 20544.931,E2 20544.931} C_VEL
LIN {X 0,Y 284.363,Z 642.815,A -85,B 0,C 180,E1 20545.986,E2 20545.986} C_VEL
LIN {X 0,Y 274.681,Z 656.933,A -85,B 0,C 180,E1 20546.769,E2 20546.769} C_VEL
LIN {X 0,Y 265.461,Z 668.704,A -85,B 0,C 180,E1 20547.521,E2 20547.521} C_VEL
LIN {X 0,Y 264.345,Z 670.289,A -85,B 0,C 180,E1 20547.735,E2 20547.735} C_VEL
LIN {X 0,Y 243.042,Z 699.106,A -85,B 0,C 180,E1 20552.75,E2 20552.75} C_VEL
LIN {X 0,Y 221.302,Z 724.239,A -85,B 0,C 180,E1 20559.672,E2 20559.672} C_VEL
LIN {X 0,Y 201.629,Z 744.444,A -85,B 0,C 180,E1 20568.661,E2 20568.661} C_VEL
LIN {X 0,Y 187.036,Z 759.158,A -85,B 0,C 180,E1 20579.683,E2 20579.683} C_VEL
LIN {X 0,Y 178.372,Z 768.792,A -85,B 0,C 180,E1 20592.716,E2 20592.716} C_VEL
LIN {X 0,Y 175.679,Z 772.746,A -85,B 0,C 180,E1 20605.056,E2 20605.056} C_VEL
LIN {X 0,Y 175.83,Z 773.08,A -85,B 0,C 180,E1 20610,E2 20610} C_VEL
LIN {X 0,Y 176.236,Z 771.651,A -85,B 0,C 180,E1 20619.894,E2 20619.894} C_VEL
LIN {X 0,Y 180.467,Z 766.206,A -85,B 0,C 180,E1 20631.621,E2 20631.621} C_VEL
LIN {X 0,Y 190.819,Z 755.221,A -85,B 0,C 180,E1 20643.742,E2 20643.742} C_VEL
LIN {X 0,Y 206.918,Z 739.096,A -85,B 0,C 180,E1 20654.041,E2 20654.041} C_VEL
LIN {X 0,Y 227.111,Z 717.686,A -85,B 0,C 180,E1 20662.345,E2 20662.345} C_VEL
LIN {X 0,Y 249.262,Z 691.03,A -85,B 0,C 180,E1 20668.764,E2 20668.764} C_VEL
LIN {X 0,Y 270.023,Z 661.303,A -85,B 0,C 180,E1 20673.352,E2 20673.352} C_VEL
LIN {X 0,Y 285.978,Z 633.635,A -85,B 0,C 180,E1 20676.308,E2 20676.308} C_VEL
LIN {X 0,Y 285.276,Z 619.157,A -85,B 0,C 180,E1 20682.235,E2 20682.235} C_VEL
LIN {X 0,Y 284.269,Z 609.957,A -85,B 0,C 180,E1 20687.702,E2 20687.702} C_VEL
LIN {X 0,Y 283.37,Z 604.122,A -85,B 0,C 180,E1 20693.868,E2 20693.868} C_VEL
LIN {X 0,Y 283.416,Z 602.68,A -85,B 0,C 180,E1 20696.94,E2 20696.94} C_VEL
LIN {X 0,Y 283.422,Z 602.953,A -85,B 0,C 180,E1 20700.002,E2 20700.002} C_VEL
LIN {X 0,Y 283.747,Z 607.747,A -85,B 0,C 180,E1 20706.127,E2 20706.127} C_VEL
LIN {X 0,Y 284.773,Z 616.998,A -85,B 0,C 180,E1 20712.28,E2 20712.28} C_VEL
LIN {X 0,Y 285.438,Z 630.77,A -85,B 0,C 180,E1 20718.158,E2 20718.158} C_VEL
LIN {X 0,Y 285.154,Z 636.209,A -85,B 0,C 180,E1 20719.878,E2 20719.878} C_VEL
LIN {X 0,Y 264.708,Z 671.374,A -85,B 0,C 180,E1 20723.765,E2 20723.765} C_VEL
LIN {X 0,Y 242.51,Z 702.69,A -85,B 0,C 180,E1 20729.061,E2 20729.061} C_VEL
LIN {X 0,Y 219.31,Z 730.87,A -85,B 0,C 180,E1 20736.621,E2 20736.621} C_VEL
LIN {X 0,Y 200.034,Z 752.613,A -85,B 0,C 180,E1 20746.041,E2 20746.041} C_VEL
LIN {X 0,Y 185.272,Z 769.431,A -85,B 0,C 180,E1 20757.912,E2 20757.912} C_VEL
LIN {X 0,Y 177.936,Z 779.637,A -85,B 0,C 180,E1 20770.1,E2 20770.1} C_VEL
LIN {X 0,Y 175.68,Z 784.283,A -85,B 0,C 180,E1 20780.074,E2 20780.074} C_VEL
LIN {X 0,Y 175.776,Z 785.866,A -85,B 0,C 180,E1 20790,E2 20790} C_VEL
LIN {X 0,Y 175.68,Z 784.297,A -85,B 0,C 180,E1 20799.926,E2 20799.926} C_VEL
LIN {X 0,Y 179.103,Z 777.779,A -85,B 0,C 180,E1 20812.717,E2 20812.717} C_VEL
LIN {X 0,Y 187.493,Z 766.765,A -85,B 0,C 180,E1 20824.423,E2 20824.423} C_VEL
LIN {X 0,Y 202.391,Z 750.051,A -85,B 0,C 180,E1 20835.332,E2 20835.332} C_VEL
LIN {X 0,Y 222.778,Z 727.01,A -85,B 0,C 180,E1 20844.646,E2 20844.646} C_VEL
LIN {X 0,Y 244.634,Z 700.043,A -85,B 0,C 180,E1 20851.481,E2 20851.481} C_VEL
LIN {X 0,Y 265.965,Z 669.521,A -85,B 0,C 180,E1 20856.516,E2 20856.516} C_VEL
LIN {X 0,Y 285.616,Z 635.134,A -85,B 0,C 180,E1 20860.349,E2 20860.349} C_VEL
LIN {X 0,Y 285.174,Z 620.901,A -85,B 0,C 180,E1 20865.92,E2 20865.92} C_VEL
LIN {X 0,Y 284.095,Z 609.866,A -85,B 0,C 180,E1 20872.342,E2 20872.342} C_VEL
LIN {X 0,Y 283.648,Z 604.878,A -85,B 0,C 180,E1 20876.939,E2 20876.939} C_VEL
LIN {X 0,Y 283.531,Z 603.228,A -85,B 0,C 180,E1 20879.998,E2 20879.998} C_VEL
LIN {X 0,Y 283.46,Z 603.112,A -85,B 0,C 180,E1 20883.06,E2 20883.06} C_VEL
LIN {X 0,Y 283.866,Z 606.689,A -85,B 0,C 180,E1 20889.205,E2 20889.205} C_VEL
LIN {X 0,Y 284.889,Z 615.103,A -85,B 0,C 180,E1 20895.407,E2 20895.407} C_VEL
LIN {X 0,Y 286.002,Z 628.622,A -85,B 0,C 180,E1 20901.747,E2 20901.747} C_VEL
LIN {X 0,Y 286.08,Z 633.819,A -85,B 0,C 180,E1 20903.62,E2 20903.62} C_VEL
LIN {X 0,Y 265.822,Z 668.1,A -85,B 0,C 180,E1 20907.409,E2 20907.409} C_VEL
LIN {X 0,Y 264.345,Z 670.289,A -85,B 0,C 180,E1 20907.735,E2 20907.735} C_VEL
LIN {X 0,Y 259.343,Z 676.848,A -85,B 0,C 180,E1 20908.451,E2 20908.451} C_VEL
LIN {X 0,Y 243.484,Z 693.743,A -85,B 0,C 180,E1 20909.985,E2 20909.985} C_VEL
LIN {X 0,Y 242.301,Z 695.178,A -85,B 0,C 180,E1 20910.248,E2 20910.248} C_VEL
LIN {X 0,Y 218.575,Z 722.145,A -85,B 0,C 180,E1 20917.19,E2 20917.19} C_VEL
LIN {X 0,Y 197.168,Z 743.361,A -85,B 0,C 180,E1 20926.279,E2 20926.279} C_VEL
LIN {X 0,Y 180.845,Z 758.814,A -85,B 0,C 180,E1 20937.713,E2 20937.713} C_VEL
LIN {X 0,Y 171.9,Z 767.742,A -85,B 0,C 180,E1 20949.37,E2 20949.37} C_VEL
LIN {X 0,Y 168.397,Z 771.986,A -85,B 0,C 180,E1 20959.64,E2 20959.64} C_VEL
LIN {X 0,Y 167.925,Z 773.367,A -85,B 0,C 180,E1 20970,E2 20970} C_VEL
LIN {X 0,Y 168.421,Z 771.941,A -85,B 0,C 180,E1 20980.358,E2 20980.358} C_VEL
LIN {X 0,Y 173.952,Z 765.546,A -85,B 0,C 180,E1 20994.097,E2 20994.097} C_VEL
LIN {X 0,Y 185.566,Z 754.231,A -85,B 0,C 180,E1 21006.268,E2 21006.268} C_VEL
LIN {X 0,Y 204.192,Z 736.514,A -85,B 0,C 180,E1 21017.076,E2 21017.076} C_VEL
LIN {X 0,Y 226.876,Z 713.009,A -85,B 0,C 180,E1 21025.449,E2 21025.449} C_VEL
LIN {X 0,Y 249.885,Z 685.324,A -85,B 0,C 180,E1 21031.471,E2 21031.471} C_VEL
LIN {X 0,Y 271.757,Z 653.494,A -85,B 0,C 180,E1 21035.833,E2 21035.833} C_VEL
LIN {X 0,Y 281.009,Z 637.466,A -85,B 0,C 180,E1 21037.466,E2 21037.466} C_VEL
LIN {X 0,Y 280.833,Z 623.782,A -85,B 0,C 180,E1 21043.501,E2 21043.501} C_VEL
LIN {X 0,Y 280.116,Z 615.302,A -85,B 0,C 180,E1 21049.098,E2 21049.098} C_VEL
LIN {X 0,Y 279.782,Z 611.247,A -85,B 0,C 180,E1 21053.789,E2 21053.789} C_VEL
LIN {X 0,Y 279.879,Z 609.798,A -85,B 0,C 180,E1 21056.901,E2 21056.901} C_VEL
LIN {X 0,Y 279.878,Z 610.068,A -85,B 0,C 180,E1 21060.002,E2 21060.002} C_VEL
LIN {X 0,Y 279.94,Z 614.935,A -85,B 0,C 180,E1 21066.211,E2 21066.211} C_VEL
LIN {X 0,Y 280.599,Z 624.568,A -85,B 0,C 180,E1 21072.465,E2 21072.465} C_VEL
LIN {X 0,Y 280.586,Z 638.969,A -85,B 0,C 180,E1 21078.554,E2 21078.554} C_VEL
LIN {X 0,Y 260.029,Z 673.136,A -85,B 0,C 180,E1 21082.423,E2 21082.423} C_VEL
LIN {X 0,Y 238.616,Z 702.338,A -85,B 0,C 180,E1 21087.331,E2 21087.331} C_VEL
LIN {X 0,Y 214.971,Z 730.022,A -85,B 0,C 180,E1 21094.66,E2 21094.66} C_VEL
LIN {X 0,Y 194.757,Z 751.729,A -85,B 0,C 180,E1 21104.02,E2 21104.02} C_VEL
LIN {X 0,Y 178.368,Z 769.129,A -85,B 0,C 180,E1 21116.511,E2 21116.511} C_VEL
LIN {X 0,Y 170.327,Z 779.34,A -85,B 0,C 180,E1 21129.171,E2 21129.171} C_VEL
LIN {X 0,Y 167.812,Z 783.991,A -85,B 0,C 180,E1 21139.604,E2 21139.604} C_VEL
LIN {X 0,Y 167.866,Z 785.578,A -85,B 0,C 180,E1 21150,E2 21150} C_VEL
LIN {X 0,Y 167.813,Z 784.006,A -85,B 0,C 180,E1 21160.396,E2 21160.396} C_VEL
LIN {X 0,Y 171.441,Z 777.71,A -85,B 0,C 180,E1 21173.418,E2 21173.418} C_VEL
LIN {X 0,Y 180.751,Z 766.462,A -85,B 0,C 180,E1 21185.901,E2 21185.901} C_VEL
LIN {X 0,Y 197.202,Z 749.08,A -85,B 0,C 180,E1 21197.403,E2 21197.403} C_VEL
LIN {X 0,Y 218.108,Z 726.685,A -85,B 0,C 180,E1 21206.414,E2 21206.414} C_VEL
LIN {X 0,Y 241.312,Z 699.053,A -85,B 0,C 180,E1 21213.322,E2 21213.322} C_VEL
LIN {X 0,Y 263.666,Z 667.816,A -85,B 0,C 180,E1 21218.306,E2 21218.306} C_VEL
LIN {X 0,Y 280.242,Z 640.081,A -85,B 0,C 180,E1 21221.302,E2 21221.302} C_VEL
LIN {X 0,Y 280.776,Z 629.567,A -85,B 0,C 180,E1 21225.238,E2 21225.238} C_VEL
LIN {X 0,Y 280.34,Z 619.307,A -85,B 0,C 180,E1 21230.675,E2 21230.675} C_VEL
LIN {X 0,Y 280.01,Z 612.019,A -85,B 0,C 180,E1 21236.899,E2 21236.899} C_VEL
LIN {X 0,Y 279.987,Z 610.335,A -85,B 0,C 180,E1 21239.998,E2 21239.998} C_VEL
LIN {X 0,Y 279.925,Z 610.212,A -85,B 0,C 180,E1 21243.099,E2 21243.099} C_VEL
LIN {X 0,Y 280.09,Z 613.926,A -85,B 0,C 180,E1 21249.33,E2 21249.33} C_VEL
LIN {X 0,Y 280.871,Z 622.567,A -85,B 0,C 180,E1 21255.633,E2 21255.633} C_VEL
LIN {X 0,Y 281.227,Z 635.996,A -85,B 0,C 180,E1 21261.858,E2 21261.858} C_VEL
LIN {X 0,Y 281.062,Z 637.829,A -85,B 0,C 180,E1 21262.508,E2 21262.508} C_VEL
LIN {X 0,Y 261.908,Z 668.945,A -85,B 0,C 180,E1 21265.929,E2 21265.929} C_VEL
LIN {X 0,Y 242.301,Z 695.178,A -85,B 0,C 180,E1 21270.248,E2 21270.248} C_VEL
LIN {X 0,Y 230.804,Z 706.608,A -85,B 0,C 180,E1 21271.884,E2 21271.884} C_VEL
LIN {X 0,Y 218.93,Z 717.12,A -85,B 0,C 180,E1 21273.8,E2 21273.8} C_VEL
LIN {X 0,Y 197.603,Z 737.997,A -85,B 0,C 180,E1 21281.661,E2 21281.661} C_VEL
LIN {X 0,Y 178.997,Z 754.663,A -85,B 0,C 180,E1 21292.173,E2 21292.173} C_VEL
LIN {X 0,Y 165.946,Z 766.577,A -85,B 0,C 180,E1 21305.82,E2 21305.82} C_VEL
LIN {X 0,Y 160.574,Z 772.275,A -85,B 0,C 180,E1 21319.13,E2 21319.13} C_VEL
LIN {X 0,Y 160.038,Z 773.654,A -85,B 0,C 180,E1 21330,E2 21330} C_VEL
LIN {X 0,Y 160.598,Z 772.231,A -85,B 0,C 180,E1 21340.869,E2 21340.869} C_VEL
LIN {X 0,Y 165.984,Z 766.482,A -85,B 0,C 180,E1 21354.209,E2 21354.209} C_VEL
LIN {X 0,Y 179.104,Z 754.528,A -85,B 0,C 180,E1 21367.8,E2 21367.8} C_VEL
LIN {X 0,Y 198.79,Z 736.823,A -85,B 0,C 180,E1 21378.778,E2 21378.778} C_VEL
LIN {X 0,Y 222.404,Z 713.342,A -85,B 0,C 180,E1 21387.156,E2 21387.156} C_VEL
LIN {X 0,Y 246.172,Z 685.674,A -85,B 0,C 180,E1 21393.107,E2 21393.107} C_VEL
LIN {X 0,Y 268.399,Z 654.246,A -85,B 0,C 180,E1 21397.343,E2 21397.343} C_VEL
LIN {X 0,Y 276.146,Z 641.054,A -85,B 0,C 180,E1 21398.769,E2 21398.769} C_VEL
LIN {X 0,Y 276.362,Z 629.659,A -85,B 0,C 180,E1 21404.105,E2 21404.105} C_VEL
LIN {X 0,Y 276.082,Z 620.415,A -85,B 0,C 180,E1 21410.819,E2 21410.819} C_VEL
LIN {X 0,Y 276.044,Z 616.759,A -85,B 0,C 180,E1 21416.858,E2 21416.858} C_VEL
LIN {X 0,Y 276.037,Z 617.018,A -85,B 0,C 180,E1 21420.002,E2 21420.002} C_VEL
LIN {X 0,Y 275.994,Z 622.081,A -85,B 0,C 180,E1 21426.3,E2 21426.3} C_VEL
LIN {X 0,Y 276.124,Z 632.012,A -85,B 0,C 180,E1 21432.671,E2 21432.671} C_VEL
LIN {X 0,Y 275.399,Z 643.492,A -85,B 0,C 180,E1 21437.482,E2 21437.482} C_VEL
LIN {X 0,Y 254.659,Z 676.102,A -85,B 0,C 180,E1 21441.209,E2 21441.209} C_VEL
LIN {X 0,Y 232.365,Z 705.032,A -85,B 0,C 180,E1 21446.205,E2 21446.205} C_VEL
LIN {X 0,Y 208.805,Z 731.291,A -85,B 0,C 180,E1 21453.365,E2 21453.365} C_VEL
LIN {X 0,Y 187.189,Z 753.224,A -85,B 0,C 180,E1 21463.281,E2 21463.281} C_VEL
LIN {X 0,Y 171.578,Z 768.829,A -85,B 0,C 180,E1 21474.998,E2 21474.998} C_VEL
LIN {X 0,Y 162.56,Z 779.344,A -85,B 0,C 180,E1 21488.649,E2 21488.649} C_VEL
LIN {X 0,Y 159.938,Z 783.699,A -85,B 0,C 180,E1 21499.086,E2 21499.086} C_VEL
LIN {X 0,Y 159.976,Z 785.292,A -85,B 0,C 180,E1 21510,E2 21510} C_VEL
LIN {X 0,Y 159.939,Z 783.714,A -85,B 0,C 180,E1 21520.914,E2 21520.914} C_VEL
LIN {X 0,Y 163.992,Z 777.413,A -85,B 0,C 180,E1 21534.55,E2 21534.55} C_VEL
LIN {X 0,Y 175.27,Z 765.025,A -85,B 0,C 180,E1 21548.481,E2 21548.481} C_VEL
LIN {X 0,Y 193.014,Z 747.459,A -85,B 0,C 180,E1 21559.894,E2 21559.894} C_VEL
LIN {X 0,Y 214.928,Z 724.998,A -85,B 0,C 180,E1 21568.67,E2 21568.67} C_VEL
LIN {X 0,Y 238.953,Z 697.138,A -85,B 0,C 180,E1 21575.406,E2 21575.406} C_VEL
LIN {X 0,Y 261.638,Z 666.114,A -85,B 0,C 180,E1 21580.12,E2 21580.12} C_VEL
LIN {X 0,Y 275.795,Z 642.697,A -85,B 0,C 180,E1 21582.739,E2 21582.739} C_VEL
LIN {X 0,Y 276.267,Z 630.546,A -85,B 0,C 180,E1 21588.139,E2 21588.139} C_VEL
LIN {X 0,Y 276.091,Z 622.311,A -85,B 0,C 180,E1 21593.702,E2 21593.702} C_VEL
LIN {X 0,Y 276.107,Z 619.06,A -85,B 0,C 180,E1 21596.855,E2 21596.855} C_VEL
LIN {X 0,Y 276.137,Z 617.284,A -85,B 0,C 180,E1 21599.998,E2 21599.998} C_VEL
LIN {X 0,Y 276.077,Z 617.169,A -85,B 0,C 180,E1 21603.142,E2 21603.142} C_VEL
LIN {X 0,Y 276.163,Z 621.094,A -85,B 0,C 180,E1 21609.464,E2 21609.464} C_VEL
LIN {X 0,Y 276.476,Z 629.977,A -85,B 0,C 180,E1 21615.888,E2 21615.888} C_VEL
LIN {X 0,Y 276.256,Z 641.53,A -85,B 0,C 180,E1 21621.29,E2 21621.29} C_VEL
LIN {X 0,Y 256.005,Z 672.842,A -85,B 0,C 180,E1 21624.847,E2 21624.847} C_VEL
LIN {X 0,Y 233.109,Z 701.63,A -85,B 0,C 180,E1 21629.864,E2 21629.864} C_VEL
LIN {X 0,Y 218.93,Z 717.12,A -85,B 0,C 180,E1 21633.8,E2 21633.8} C_VEL
LIN {X 0,Y 206.95,Z 726.909,A -85,B 0,C 180,E1 21636.069,E2 21636.069} C_VEL
LIN {X 0,Y 195.095,Z 735.815,A -85,B 0,C 180,E1 21638.709,E2 21638.709} C_VEL
LIN {X 0,Y 174.372,Z 753.52,A -85,B 0,C 180,E1 21649.364,E2 21649.364} C_VEL
LIN {X 0,Y 160.605,Z 765.089,A -85,B 0,C 180,E1 21661.876,E2 21661.876} C_VEL
LIN {X 0,Y 154.446,Z 770.807,A -85,B 0,C 180,E1 21672.896,E2 21672.896} C_VEL
LIN {X 0,Y 151.972,Z 773.684,A -85,B 0,C 180,E1 21684.969,E2 21684.969} C_VEL
LIN {X 0,Y 152.005,Z 773.664,A -85,B 0,C 180,E1 21695.169,E2 21695.169} C_VEL
LIN {X 0,Y 155.615,Z 769.602,A -85,B 0,C 180,E1 21709.911,E2 21709.911} C_VEL
LIN {X 0,Y 166.831,Z 759.784,A -85,B 0,C 180,E1 21724.666,E2 21724.666} C_VEL
LIN {X 0,Y 185.961,Z 743.787,A -85,B 0,C 180,E1 21737.122,E2 21737.122} C_VEL
LIN {X 0,Y 209.318,Z 722.531,A -85,B 0,C 180,E1 21746.292,E2 21746.292} C_VEL
LIN {X 0,Y 234.428,Z 695.932,A -85,B 0,C 180,E1 21752.999,E2 21752.999} C_VEL
LIN {X 0,Y 257.623,Z 666.25,A -85,B 0,C 180,E1 21757.609,E2 21757.609} C_VEL
LIN {X 0,Y 271.309,Z 645.251,A -85,B 0,C 180,E1 21759.91,E2 21759.91} C_VEL
LIN {X 0,Y 271.929,Z 634.219,A -85,B 0,C 180,E1 21765.493,E2 21765.493} C_VEL
LIN {X 0,Y 271.966,Z 626.35,A -85,B 0,C 180,E1 21771.841,E2 21771.841} C_VEL
LIN {X 0,Y 272.146,Z 623.683,A -85,B 0,C 180,E1 21776.813,E2 21776.813} C_VEL
LIN {X 0,Y 272.135,Z 623.928,A -85,B 0,C 180,E1 21780.002,E2 21780.002} C_VEL
LIN {X 0,Y 271.786,Z 629.059,A -85,B 0,C 180,E1 21786.398,E2 21786.398} C_VEL
LIN {X 0,Y 271.561,Z 637.802,A -85,B 0,C 180,E1 21792.069,E2 21792.069} C_VEL
LIN {X 0,Y 270.418,Z 647.619,A -85,B 0,C 180,E1 21796.258,E2 21796.258} C_VEL
LIN {X 0,Y 247.174,Z 682.098,A -85,B 0,C 180,E1 21800.359,E2 21800.359} C_VEL
LIN {X 0,Y 221.847,Z 712.663,A -85,B 0,C 180,E1 21806.149,E2 21806.149} C_VEL
LIN {X 0,Y 197.826,Z 737.577,A -85,B 0,C 180,E1 21813.903,E2 21813.903} C_VEL
LIN {X 0,Y 175.518,Z 758.553,A -85,B 0,C 180,E1 21824.999,E2 21824.999} C_VEL
LIN {X 0,Y 160.64,Z 772.729,A -85,B 0,C 180,E1 21838.023,E2 21838.023} C_VEL
LIN {X 0,Y 153.25,Z 781.463,A -85,B 0,C 180,E1 21852.758,E2 21852.758} C_VEL
LIN {X 0,Y 151.733,Z 784.755,A -85,B 0,C 180,E1 21866.224,E2 21866.224} C_VEL
LIN {X 0,Y 151.728,Z 784.76,A -85,B 0,C 180,E1 21873.745,E2 21873.745} C_VEL
LIN {X 0,Y 153.248,Z 781.486,A -85,B 0,C 180,E1 21887.242,E2 21887.242} C_VEL
LIN {X 0,Y 160.599,Z 772.785,A -85,B 0,C 180,E1 21901.954,E2 21901.954} C_VEL
LIN {X 0,Y 176.912,Z 757.356,A -85,B 0,C 180,E1 21915.911,E2 21915.911} C_VEL
LIN {X 0,Y 199.314,Z 736.198,A -85,B 0,C 180,E1 21926.682,E2 21926.682} C_VEL
LIN {X 0,Y 224.041,Z 710.47,A -85,B 0,C 180,E1 21934.36,E2 21934.36} C_VEL
LIN {X 0,Y 248.345,Z 680.681,A -85,B 0,C 180,E1 21939.885,E2 21939.885} C_VEL
LIN {X 0,Y 270.597,Z 647.629,A -85,B 0,C 180,E1 21943.753,E2 21943.753} C_VEL
LIN {X 0,Y 271.702,Z 637.897,A -85,B 0,C 180,E1 21947.937,E2 21947.937} C_VEL
LIN {X 0,Y 271.883,Z 629.27,A -85,B 0,C 180,E1 21953.604,E2 21953.604} C_VEL
LIN {X 0,Y 272.075,Z 626.006,A -85,B 0,C 180,E1 21956.808,E2 21956.808} C_VEL
LIN {X 0,Y 272.225,Z 624.188,A -85,B 0,C 180,E1 21959.998,E2 21959.998} C_VEL
LIN {X 0,Y 272.158,Z 624.09,A -85,B 0,C 180,E1 21963.187,E2 21963.187} C_VEL
LIN {X 0,Y 271.981,Z 628.111,A -85,B 0,C 180,E1 21969.611,E2 21969.611} C_VEL
LIN {X 0,Y 271.899,Z 637.373,A -85,B 0,C 180,E1 21976.163,E2 21976.163} C_VEL
LIN {X 0,Y 271.386,Z 645.539,A -85,B 0,C 180,E1 21980.051,E2 21980.051} C_VEL
LIN {X 0,Y 248.604,Z 678.822,A -85,B 0,C 180,E1 21983.995,E2 21983.995} C_VEL
LIN {X 0,Y 223.933,Z 707.824,A -85,B 0,C 180,E1 21989.477,E2 21989.477} C_VEL
LIN {X 0,Y 200.196,Z 731.277,A -85,B 0,C 180,E1 21996.775,E2 21996.775} C_VEL
LIN {X 0,Y 195.095,Z 735.815,A -85,B 0,C 180,E1 21998.709,E2 21998.709} C_VEL
LIN {X 0,Y 183.332,Z 743.952,A -85,B 0,C 180,E1 22001.792,E2 22001.792} C_VEL
LIN {X 0,Y 171.874,Z 751.037,A -85,B 0,C 180,E1 22005.415,E2 22005.415} C_VEL
LIN {X 0,Y 155.962,Z 763.54,A -85,B 0,C 180,E1 22017.727,E2 22017.727} C_VEL
LIN {X 0,Y 146.816,Z 771.097,A -85,B 0,C 180,E1 22031.977,E2 22031.977} C_VEL
LIN {X 0,Y 144.126,Z 773.898,A -85,B 0,C 180,E1 22043.97,E2 22043.97} C_VEL
LIN {X 0,Y 144.245,Z 774.229,A -85,B 0,C 180,E1 22050,E2 22050} C_VEL
LIN {X 0,Y 145.01,Z 772.81,A -85,B 0,C 180,E1 22062.054,E2 22062.054} C_VEL
LIN {X 0,Y 151.652,Z 766.918,A -85,B 0,C 180,E1 22076.989,E2 22076.989} C_VEL
LIN {X 0,Y 166.622,Z 755.12,A -85,B 0,C 180,E1 22091.21,E2 22091.21} C_VEL
LIN {X 0,Y 188.513,Z 737.443,A -85,B 0,C 180,E1 22102.482,E2 22102.482} C_VEL
LIN {X 0,Y 214.514,Z 713.598,A -85,B 0,C 180,E1 22110.866,E2 22110.866} C_VEL
LIN {X 0,Y 239.362,Z 686.39,A -85,B 0,C 180,E1 22116.524,E2 22116.524} C_VEL
LIN {X 0,Y 262.337,Z 655.62,A -85,B 0,C 180,E1 22120.489,E2 22120.489} C_VEL
LIN {X 0,Y 266.086,Z 649.804,A -85,B 0,C 180,E1 22121.064,E2 22121.064} C_VEL
LIN {X 0,Y 267.225,Z 641.376,A -85,B 0,C 180,E1 22125.23,E2 22125.23} C_VEL
LIN {X 0,Y 267.738,Z 633.147,A -85,B 0,C 180,E1 22131.875,E2 22131.875} C_VEL
LIN {X 0,Y 267.971,Z 630.468,A -85,B 0,C 180,E1 22136.763,E2 22136.763} C_VEL
LIN {X 0,Y 267.956,Z 630.708,A -85,B 0,C 180,E1 22140.002,E2 22140.002} C_VEL
LIN {X 0,Y 267.481,Z 636.026,A -85,B 0,C 180,E1 22146.502,E2 22146.502} C_VEL
LIN {X 0,Y 266.686,Z 645.675,A -85,B 0,C 180,E1 22152.604,E2 22152.604} C_VEL
LIN {X 0,Y 266.121,Z 650.166,A -85,B 0,C 180,E1 22154.706,E2 22154.706} C_VEL
LIN {X 0,Y 242.763,Z 683.824,A -85,B 0,C 180,E1 22158.875,E2 22158.875} C_VEL
LIN {X 0,Y 218.032,Z 712.653,A -85,B 0,C 180,E1 22164.29,E2 22164.29} C_VEL
LIN {X 0,Y 192.463,Z 738.008,A -85,B 0,C 180,E1 22172.163,E2 22172.163} C_VEL
LIN {X 0,Y 169.664,Z 758.345,A -85,B 0,C 180,E1 22183.099,E2 22183.099} C_VEL
LIN {X 0,Y 153.72,Z 772.429,A -85,B 0,C 180,E1 22196.398,E2 22196.398} C_VEL
LIN {X 0,Y 145.563,Z 781.168,A -85,B 0,C 180,E1 22211.817,E2 22211.817} C_VEL
LIN {X 0,Y 143.862,Z 784.301,A -85,B 0,C 180,E1 22223.958,E2 22223.958} C_VEL
LIN {X 0,Y 144.153,Z 784.716,A -85,B 0,C 180,E1 22230,E2 22230} C_VEL
LIN {X 0,Y 144.253,Z 783.132,A -85,B 0,C 180,E1 22242.118,E2 22242.118} C_VEL
LIN {X 0,Y 149.279,Z 776.82,A -85,B 0,C 180,E1 22257.157,E2 22257.157} C_VEL
LIN {X 0,Y 163.118,Z 764.042,A -85,B 0,C 180,E1 22272.448,E2 22272.448} C_VEL
LIN {X 0,Y 183.965,Z 745.834,A -85,B 0,C 180,E1 22284.367,E2 22284.367} C_VEL
LIN {X 0,Y 209.226,Z 721.918,A -85,B 0,C 180,E1 22293.332,E2 22293.332} C_VEL
LIN {X 0,Y 236.027,Z 692.43,A -85,B 0,C 180,E1 22299.804,E2 22299.804} C_VEL
LIN {X 0,Y 261.126,Z 658.628,A -85,B 0,C 180,E1 22304.31,E2 22304.31} C_VEL
LIN {X 0,Y 266.217,Z 650.455,A -85,B 0,C 180,E1 22305.215,E2 22305.215} C_VEL
LIN {X 0,Y 267.325,Z 639.484,A -85,B 0,C 180,E1 22311.038,E2 22311.038} C_VEL
LIN {X 0,Y 267.841,Z 632.892,A -85,B 0,C 180,E1 22316.758,E2 22316.758} C_VEL
LIN {X 0,Y 268.067,Z 630.937,A -85,B 0,C 180,E1 22319.998,E2 22319.998} C_VEL
LIN {X 0,Y 267.994,Z 630.86,A -85,B 0,C 180,E1 22323.237,E2 22323.237} C_VEL
LIN {X 0,Y 267.697,Z 635.107,A -85,B 0,C 180,E1 22329.766,E2 22329.766} C_VEL
LIN {X 0,Y 267.209,Z 643.093,A -85,B 0,C 180,E1 22335.57,E2 22335.57} C_VEL
LIN {X 0,Y 266.069,Z 650.12,A -85,B 0,C 180,E1 22338.858,E2 22338.858} C_VEL
LIN {X 0,Y 243.916,Z 681.06,A -85,B 0,C 180,E1 22342.574,E2 22342.574} C_VEL
LIN {X 0,Y 220.071,Z 708.143,A -85,B 0,C 180,E1 22347.647,E2 22347.647} C_VEL
LIN {X 0,Y 195.944,Z 731.186,A -85,B 0,C 180,E1 22354.719,E2 22354.719} C_VEL
LIN {X 0,Y 172.122,Z 750.849,A -85,B 0,C 180,E1 22365.272,E2 22365.272} C_VEL
LIN {X 0,Y 171.874,Z 751.037,A -85,B 0,C 180,E1 22365.415,E2 22365.415} C_VEL
LIN {X 0,Y 160.924,Z 757.286,A -85,B 0,C 180,E1 22369.634,E2 22369.634} C_VEL
LIN {X 0,Y 150.783,Z 762.622,A -85,B 0,C 180,E1 22374.508,E2 22374.508} C_VEL
LIN {X 0,Y 140.632,Z 770.243,A -85,B 0,C 180,E1 22387.862,E2 22387.862} C_VEL
LIN {X 0,Y 136.257,Z 774.186,A -85,B 0,C 180,E1 22403.62,E2 22403.62} C_VEL
LIN {X 0,Y 136.258,Z 774.485,A -85,B 0,C 180,E1 22410.715,E2 22410.715} C_VEL
LIN {X 0,Y 137.253,Z 773.099,A -85,B 0,C 180,E1 22422.746,E2 22422.746} C_VEL
LIN {X 0,Y 144.326,Z 767.345,A -85,B 0,C 180,E1 22438.171,E2 22438.171} C_VEL
LIN {X 0,Y 160.645,Z 755.415,A -85,B 0,C 180,E1 22453.105,E2 22453.105} C_VEL
LIN {X 0,Y 183.71,Z 737.75,A -85,B 0,C 180,E1 22464.479,E2 22464.479} C_VEL
LIN {X 0,Y 210.715,Z 713.923,A -85,B 0,C 180,E1 22472.777,E2 22472.777} C_VEL
LIN {X 0,Y 236.296,Z 686.745,A -85,B 0,C 180,E1 22478.3,E2 22478.3} C_VEL
LIN {X 0,Y 259.939,Z 655.816,A -85,B 0,C 180,E1 22482.159,E2 22482.159} C_VEL
LIN {X 0,Y 261.714,Z 652.602,A -85,B 0,C 180,E1 22482.737,E2 22482.737} C_VEL
LIN {X 0,Y 262.878,Z 643.657,A -85,B 0,C 180,E1 22488.286,E2 22488.286} C_VEL
LIN {X 0,Y 263.385,Z 638.72,A -85,B 0,C 180,E1 22493.4,E2 22493.4} C_VEL
LIN {X 0,Y 263.688,Z 637.19,A -85,B 0,C 180,E1 22496.71,E2 22496.71} C_VEL
LIN {X 0,Y 263.403,Z 638.392,A -85,B 0,C 180,E1 22501.649,E2 22501.649} C_VEL
LIN {X 0,Y 262.767,Z 643.956,A -85,B 0,C 180,E1 22507.497,E2 22507.497} C_VEL
LIN {X 0,Y 261.35,Z 654.039,A -85,B 0,C 180,E1 22513.4,E2 22513.4} C_VEL
LIN {X 0,Y 238.034,Z 686.13,A -85,B 0,C 180,E1 22517.417,E2 22517.417} C_VEL
LIN {X 0,Y 212.133,Z 714.954,A -85,B 0,C 180,E1 22522.918,E2 22522.918} C_VEL
LIN {X 0,Y 186.769,Z 738.903,A -85,B 0,C 180,E1 22530.529,E2 22530.529} C_VEL
LIN {X 0,Y 164.694,Z 757.579,A -85,B 0,C 180,E1 22540.639,E2 22540.639} C_VEL
LIN {X 0,Y 147.013,Z 772.079,A -85,B 0,C 180,E1 22554.553,E2 22554.553} C_VEL
LIN {X 0,Y 137.898,Z 780.873,A -85,B 0,C 180,E1 22570.767,E2 22570.767} C_VEL
LIN {X 0,Y 135.944,Z 784.011,A -85,B 0,C 180,E1 22583.605,E2 22583.605} C_VEL
LIN {X 0,Y 136.264,Z 784.429,A -85,B 0,C 180,E1 22590,E2 22590} C_VEL
LIN {X 0,Y 136.443,Z 782.841,A -85,B 0,C 180,E1 22602.823,E2 22602.823} C_VEL
LIN {X 0,Y 142.053,Z 776.524,A -85,B 0,C 180,E1 22618.663,E2 22618.663} C_VEL
LIN {X 0,Y 156.962,Z 763.857,A -85,B 0,C 180,E1 22634.377,E2 22634.377} C_VEL
LIN {X 0,Y 179.29,Z 745.528,A -85,B 0,C 180,E1 22646.508,E2 22646.508} C_VEL
LIN {X 0,Y 205.324,Z 721.898,A -85,B 0,C 180,E1 22655.306,E2 22655.306} C_VEL
LIN {X 0,Y 231.698,Z 693.926,A -85,B 0,C 180,E1 22661.378,E2 22661.378} C_VEL
LIN {X 0,Y 256.903,Z 661.299,A -85,B 0,C 180,E1 22665.731,E2 22665.731} C_VEL
LIN {X 0,Y 261.452,Z 654.176,A -85,B 0,C 180,E1 22666.606,E2 22666.606} C_VEL
LIN {X 0,Y 262.74,Z 645.462,A -85,B 0,C 180,E1 22671.547,E2 22671.547} C_VEL
LIN {X 0,Y 263.399,Z 639.654,A -85,B 0,C 180,E1 22676.703,E2 22676.703} C_VEL
LIN {X 0,Y 263.783,Z 637.626,A -85,B 0,C 180,E1 22679.998,E2 22679.998} C_VEL
LIN {X 0,Y 263.699,Z 637.563,A -85,B 0,C 180,E1 22683.289,E2 22683.289} C_VEL
LIN {X 0,Y 263.246,Z 640.682,A -85,B 0,C 180,E1 22688.68,E2 22688.68} C_VEL
LIN {X 0,Y 262.41,Z 648.891,A -85,B 0,C 180,E1 22695.068,E2 22695.068} C_VEL
LIN {X 0,Y 261.858,Z 652.796,A -85,B 0,C 180,E1 22697.233,E2 22697.233} C_VEL
LIN {X 0,Y 250.55,Z 669.183,A -85,B 0,C 180,E1 22699.17,E2 22699.17} C_VEL
LIN {X 0,Y 225.547,Z 699.043,A -85,B 0,C 180,E1 22703.747,E2 22703.747} C_VEL
LIN {X 0,Y 198.757,Z 725.112,A -85,B 0,C 180,E1 22710.414,E2 22710.414} C_VEL
LIN {X 0,Y 173.621,Z 745.743,A -85,B 0,C 180,E1 22719.694,E2 22719.694} C_VEL
LIN {X 0,Y 153.44,Z 760.679,A -85,B 0,C 180,E1 22732.118,E2 22732.118} C_VEL
LIN {X 0,Y 150.783,Z 762.622,A -85,B 0,C 180,E1 22734.508,E2 22734.508} C_VEL
LIN {X 0,Y 146.672,Z 764.953,A -85,B 0,C 180,E1 22737.347,E2 22737.347} C_VEL
LIN {X 0,Y 133.877,Z 770.154,A -85,B 0,C 180,E1 22745.518,E2 22745.518} C_VEL
LIN {X 0,Y 133.309,Z 770.461,A -85,B 0,C 180,E1 22746.415,E2 22746.415} C_VEL
LIN {X 0,Y 128.376,Z 774.474,A -85,B 0,C 180,E1 22763.227,E2 22763.227} C_VEL
LIN {X 0,Y 128.458,Z 774.803,A -85,B 0,C 180,E1 22770,E2 22770} C_VEL
LIN {X 0,Y 129.487,Z 773.39,A -85,B 0,C 180,E1 22783.525,E2 22783.525} C_VEL
LIN {X 0,Y 137.3,Z 767.637,A -85,B 0,C 180,E1 22799.753,E2 22799.753} C_VEL
LIN {X 0,Y 154.851,Z 755.709,A -85,B 0,C 180,E1 22815.146,E2 22815.146} C_VEL
LIN {X 0,Y 179.105,Z 738.086,A -85,B 0,C 180,E1 22826.567,E2 22826.567} C_VEL
LIN {X 0,Y 207.172,Z 714.245,A -85,B 0,C 180,E1 22834.748,E2 22834.748} C_VEL
LIN {X 0,Y 233.455,Z 687.102,A -85,B 0,C 180,E1 22840.126,E2 22840.126} C_VEL
LIN {X 0,Y 256.129,Z 658.349,A -85,B 0,C 180,E1 22843.637,E2 22843.637} C_VEL
LIN {X 0,Y 257.483,Z 653.923,A -85,B 0,C 180,E1 22845.678,E2 22845.678} C_VEL
LIN {X 0,Y 258.604,Z 647.048,A -85,B 0,C 180,E1 22851.228,E2 22851.228} C_VEL
LIN {X 0,Y 259.223,Z 643.762,A -85,B 0,C 180,E1 22856.654,E2 22856.654} C_VEL
LIN {X 0,Y 258.915,Z 644.992,A -85,B 0,C 180,E1 22861.677,E2 22861.677} C_VEL
LIN {X 0,Y 257.955,Z 650.756,A -85,B 0,C 180,E1 22867.638,E2 22867.638} C_VEL
LIN {X 0,Y 256.282,Z 658.825,A -85,B 0,C 180,E1 22872.278,E2 22872.278} C_VEL
LIN {X 0,Y 230.807,Z 691.616,A -85,B 0,C 180,E1 22876.377,E2 22876.377} C_VEL
LIN {X 0,Y 202.084,Z 721.378,A -85,B 0,C 180,E1 22882.544,E2 22882.544} C_VEL
LIN {X 0,Y 176.132,Z 744.125,A -85,B 0,C 180,E1 22890.721,E2 22890.721} C_VEL
LIN {X 0,Y 153.139,Z 762.076,A -85,B 0,C 180,E1 22902.136,E2 22902.136} C_VEL
LIN {X 0,Y 137.129,Z 774.339,A -85,B 0,C 180,E1 22916.49,E2 22916.49} C_VEL
LIN {X 0,Y 130.278,Z 780.577,A -85,B 0,C 180,E1 22929.594,E2 22929.594} C_VEL
LIN {X 0,Y 128.028,Z 783.72,A -85,B 0,C 180,E1 22943.208,E2 22943.208} C_VEL
LIN {X 0,Y 128.345,Z 784.141,A -85,B 0,C 180,E1 22950,E2 22950} C_VEL
LIN {X 0,Y 128.62,Z 782.549,A -85,B 0,C 180,E1 22963.618,E2 22963.618} C_VEL
LIN {X 0,Y 134.922,Z 776.227,A -85,B 0,C 180,E1 22980.331,E2 22980.331} C_VEL
LIN {X 0,Y 151.162,Z 763.556,A -85,B 0,C 180,E1 22996.569,E2 22996.569} C_VEL
LIN {X 0,Y 174.444,Z 745.537,A -85,B 0,C 180,E1 23008.616,E2 23008.616} C_VEL
LIN {X 0,Y 200.239,Z 723.201,A -85,B 0,C 180,E1 23016.977,E2 23016.977} C_VEL
LIN {X 0,Y 227.077,Z 695.93,A -85,B 0,C 180,E1 23022.933,E2 23022.933} C_VEL
LIN {X 0,Y 252.009,Z 665.06,A -85,B 0,C 180,E1 23027.07,E2 23027.07} C_VEL
LIN {X 0,Y 256.327,Z 659.089,A -85,B 0,C 180,E1 23027.69,E2 23027.69} C_VEL
LIN {X 0,Y 258.039,Z 650.985,A -85,B 0,C 180,E1 23032.326,E2 23032.326} C_VEL
LIN {X 0,Y 259.039,Z 645.175,A -85,B 0,C 180,E1 23038.324,E2 23038.324} C_VEL
LIN {X 0,Y 259.228,Z 644.145,A -85,B 0,C 180,E1 23043.346,E2 23043.346} C_VEL
LIN {X 0,Y 258.629,Z 647.439,A -85,B 0,C 180,E1 23048.836,E2 23048.836} C_VEL
LIN {X 0,Y 257.359,Z 655.377,A -85,B 0,C 180,E1 23055.004,E2 23055.004} C_VEL
LIN {X 0,Y 256.388,Z 658.249,A -85,B 0,C 180,E1 23056.231,E2 23056.231} C_VEL
LIN {X 0,Y 231.803,Z 689.262,A -85,B 0,C 180,E1 23060.12,E2 23060.12} C_VEL
LIN {X 0,Y 204.12,Z 717.223,A -85,B 0,C 180,E1 23065.919,E2 23065.919} C_VEL
LIN {X 0,Y 177.626,Z 739.303,A -85,B 0,C 180,E1 23073.916,E2 23073.916} C_VEL
LIN {X 0,Y 154.746,Z 755.835,A -85,B 0,C 180,E1 23084.815,E2 23084.815} C_VEL
LIN {X 0,Y 137.272,Z 767.708,A -85,B 0,C 180,E1 23100.241,E2 23100.241} C_VEL
LIN {X 0,Y 133.309,Z 770.461,A -85,B 0,C 180,E1 23106.415,E2 23106.415} C_VEL
LIN {X 0,Y 128.384,Z 772.446,A -85,B 0,C 180,E1 23111.684,E2 23111.684} C_VEL
LIN {X 0,Y 120.835,Z 774.407,A -85,B 0,C 180,E1 23120.137,E2 23120.137} C_VEL
LIN {X 0,Y 120.626,Z 774.531,A -85,B 0,C 180,E1 23121.178,E2 23121.178} C_VEL
LIN {X 0,Y 120.548,Z 775.09,A -85,B 0,C 180,E1 23130,E2 23130} C_VEL
LIN {X 0,Y 121.761,Z 773.68,A -85,B 0,C 180,E1 23144.401,E2 23144.401} C_VEL
LIN {X 0,Y 130.369,Z 767.929,A -85,B 0,C 180,E1 23161.51,E2 23161.51} C_VEL
LIN {X 0,Y 149.233,Z 756.023,A -85,B 0,C 180,E1 23177.325,E2 23177.325} C_VEL
LIN {X 0,Y 174.314,Z 738.744,A -85,B 0,C 180,E1 23188.596,E2 23188.596} C_VEL
LIN {X 0,Y 202.345,Z 715.993,A -85,B 0,C 180,E1 23196.443,E2 23196.443} C_VEL
LIN {X 0,Y 230.866,Z 687.458,A -85,B 0,C 180,E1 23201.987,E2 23201.987} C_VEL
LIN {X 0,Y 251.714,Z 661.801,A -85,B 0,C 180,E1 23205.061,E2 23205.061} C_VEL
LIN {X 0,Y 253.455,Z 655.046,A -85,B 0,C 180,E1 23209.679,E2 23209.679} C_VEL
LIN {X 0,Y 254.094,Z 651.922,A -85,B 0,C 180,E1 23213.158,E2 23213.158} C_VEL
LIN {X 0,Y 254.585,Z 650.235,A -85,B 0,C 180,E1 23216.593,E2 23216.593} C_VEL
LIN {X 0,Y 254.219,Z 651.455,A -85,B 0,C 180,E1 23221.708,E2 23221.708} C_VEL
LIN {X 0,Y 252.972,Z 657.429,A -85,B 0,C 180,E1 23227.741,E2 23227.741} C_VEL
LIN {X 0,Y 252.019,Z 661.496,A -85,B 0,C 180,E1 23230.384,E2 23230.384} C_VEL
LIN {X 0,Y 249.547,Z 665.399,A -85,B 0,C 180,E1 23231.183,E2 23231.183} C_VEL
LIN {X 0,Y 223.651,Z 696.632,A -85,B 0,C 180,E1 23235.261,E2 23235.261} C_VEL
LIN {X 0,Y 196.829,Z 723.036,A -85,B 0,C 180,E1 23240.9,E2 23240.9} C_VEL
LIN {X 0,Y 169.591,Z 745.651,A -85,B 0,C 180,E1 23249.258,E2 23249.258} C_VEL
LIN {X 0,Y 145.621,Z 763.191,A -85,B 0,C 180,E1 23261.076,E2 23261.076} C_VEL
LIN {X 0,Y 127.913,Z 775.895,A -85,B 0,C 180,E1 23277.814,E2 23277.814} C_VEL
LIN {X 0,Y 120.819,Z 782.237,A -85,B 0,C 180,E1 23295.484,E2 23295.484} C_VEL
LIN {X 0,Y 120.433,Z 783.854,A -85,B 0,C 180,E1 23310,E2 23310} C_VEL
LIN {X 0,Y 120.818,Z 782.256,A -85,B 0,C 180,E1 23324.516,E2 23324.516} C_VEL
LIN {X 0,Y 127.917,Z 775.93,A -85,B 0,C 180,E1 23342.185,E2 23342.185} C_VEL
LIN {X 0,Y 145.615,Z 763.256,A -85,B 0,C 180,E1 23358.927,E2 23358.927} C_VEL
LIN {X 0,Y 169.613,Z 745.73,A -85,B 0,C 180,E1 23370.746,E2 23370.746} C_VEL
LIN {X 0,Y 196.929,Z 723.092,A -85,B 0,C 180,E1 23379.116,E2 23379.116} C_VEL
LIN {X 0,Y 223.667,Z 696.828,A -85,B 0,C 180,E1 23384.723,E2 23384.723} C_VEL
LIN {X 0,Y 249.685,Z 665.513,A -85,B 0,C 180,E1 23388.806,E2 23388.806} C_VEL
LIN {X 0,Y 251.08,Z 663.625,A -85,B 0,C 180,E1 23388.995,E2 23388.995} C_VEL
LIN {X 0,Y 252.525,Z 660.146,A -85,B 0,C 180,E1 23390.508,E2 23390.508} C_VEL
LIN {X 0,Y 254.035,Z 652.869,A -85,B 0,C 180,E1 23396.581,E2 23396.581} C_VEL
LIN {X 0,Y 254.656,Z 650.667,A -85,B 0,C 180,E1 23399.998,E2 23399.998} C_VEL
LIN {X 0,Y 254.569,Z 650.611,A -85,B 0,C 180,E1 23403.408,E2 23403.408} C_VEL
LIN {X 0,Y 253.842,Z 653.611,A -85,B 0,C 180,E1 23408.573,E2 23408.573} C_VEL
LIN {X 0,Y 252.233,Z 661.167,A -85,B 0,C 180,E1 23414.602,E2 23414.602} C_VEL
LIN {X 0,Y 227.543,Z 691.324,A -85,B 0,C 180,E1 23418.516,E2 23418.516} C_VEL
LIN {X 0,Y 200.738,Z 717.533,A -85,B 0,C 180,E1 23423.856,E2 23423.856} C_VEL
LIN {X 0,Y 173.809,Z 739.208,A -85,B 0,C 180,E1 23431.505,E2 23431.505} C_VEL
LIN {X 0,Y 149.048,Z 756.191,A -85,B 0,C 180,E1 23442.671,E2 23442.671} C_VEL
LIN {X 0,Y 130.339,Z 768,A -85,B 0,C 180,E1 23458.482,E2 23458.482} C_VEL
LIN {X 0,Y 121.745,Z 773.72,A -85,B 0,C 180,E1 23475.597,E2 23475.597} C_VEL
LIN {X 0,Y 120.626,Z 774.531,A -85,B 0,C 180,E1 23481.178,E2 23481.178} C_VEL
LIN {X 0,Y 117.787,Z 775.238,A -85,B 0,C 180,E1 23487.326,E2 23487.326} C_VEL
LIN {X 0,Y 112.689,Z 774.97,A -85,B 0,C 180,E1 23498.139,E2 23498.139} C_VEL
LIN {X 0,Y 119.052,Z 770.867,A -85,B 0,C 180,E1 23517.115,E2 23517.115} C_VEL
LIN {X 0,Y 135.421,Z 761.332,A -85,B 0,C 180,E1 23534.332,E2 23534.332} C_VEL
LIN {X 0,Y 161.209,Z 745.288,A -85,B 0,C 180,E1 23547.706,E2 23547.706} C_VEL
LIN {X 0,Y 190.558,Z 723.604,A -85,B 0,C 180,E1 23556.597,E2 23556.597} C_VEL
LIN {X 0,Y 220.174,Z 696.603,A -85,B 0,C 180,E1 23562.536,E2 23562.536} C_VEL
LIN {X 0,Y 246.65,Z 666.344,A -85,B 0,C 180,E1 23566.416,E2 23566.416} C_VEL
LIN {X 0,Y 247.805,Z 663.577,A -85,B 0,C 180,E1 23567.858,E2 23567.858} C_VEL
LIN {X 0,Y 249.23,Z 658.414,A -85,B 0,C 180,E1 23573.024,E2 23573.024} C_VEL
LIN {X 0,Y 249.806,Z 656.63,A -85,B 0,C 180,E1 23576.527,E2 23576.527} C_VEL
LIN {X 0,Y 249.431,Z 657.854,A -85,B 0,C 180,E1 23581.741,E2 23581.741} C_VEL
LIN {X 0,Y 247.693,Z 664.137,A -85,B 0,C 180,E1 23587.999,E2 23587.999} C_VEL
LIN {X 0,Y 246.607,Z 666.978,A -85,B 0,C 180,E1 23589.527,E2 23589.527} C_VEL
LIN {X 0,Y 219.944,Z 698.066,A -85,B 0,C 180,E1 23593.494,E2 23593.494} C_VEL
LIN {X 0,Y 192.221,Z 724.277,A -85,B 0,C 180,E1 23599.047,E2 23599.047} C_VEL
LIN {X 0,Y 165.447,Z 745.529,A -85,B 0,C 180,E1 23606.856,E2 23606.856} C_VEL
LIN {X 0,Y 140.318,Z 762.887,A -85,B 0,C 180,E1 23618.526,E2 23618.526} C_VEL
LIN {X 0,Y 123.768,Z 773.738,A -85,B 0,C 180,E1 23632.288,E2 23632.288} C_VEL
LIN {X 0,Y 115.181,Z 780.042,A -85,B 0,C 180,E1 23646.95,E2 23646.95} C_VEL
LIN {X 0,Y 112.222,Z 783.14,A -85,B 0,C 180,E1 23662.246,E2 23662.246} C_VEL
LIN {X 0,Y 112.511,Z 783.566,A -85,B 0,C 180,E1 23670,E2 23670} C_VEL
LIN {X 0,Y 113.047,Z 781.964,A -85,B 0,C 180,E1 23685.538,E2 23685.538} C_VEL
LIN {X 0,Y 120.996,Z 775.687,A -85,B 0,C 180,E1 23704.134,E2 23704.134} C_VEL
LIN {X 0,Y 140.309,Z 762.953,A -85,B 0,C 180,E1 23721.479,E2 23721.479} C_VEL
LIN {X 0,Y 166.868,Z 744.611,A -85,B 0,C 180,E1 23733.636,E2 23733.636} C_VEL
LIN {X 0,Y 196.813,Z 720.519,A -85,B 0,C 180,E1 23741.962,E2 23741.962} C_VEL
LIN {X 0,Y 226.741,Z 691.105,A -85,B 0,C 180,E1 23747.588,E2 23747.588} C_VEL
LIN {X 0,Y 247.19,Z 666.391,A -85,B 0,C 180,E1 23750.625,E2 23750.625} C_VEL
LIN {X 0,Y 249.127,Z 659.364,A -85,B 0,C 180,E1 23756.514,E2 23756.514} C_VEL
LIN {X 0,Y 249.878,Z 657.047,A -85,B 0,C 180,E1 23759.998,E2 23759.998} C_VEL
LIN {X 0,Y 249.793,Z 657.001,A -85,B 0,C 180,E1 23763.473,E2 23763.473} C_VEL
LIN {X 0,Y 248.718,Z 660.573,A -85,B 0,C 180,E1 23769.211,E2 23769.211} C_VEL
LIN {X 0,Y 247.073,Z 666.032,A -85,B 0,C 180,E1 23773.417,E2 23773.417} C_VEL
LIN {X 0,Y 219.89,Z 697.12,A -85,B 0,C 180,E1 23777.445,E2 23777.445} C_VEL
LIN {X 0,Y 191.946,Z 722.58,A -85,B 0,C 180,E1 23782.991,E2 23782.991} C_VEL
LIN {X 0,Y 162.994,Z 744.165,A -85,B 0,C 180,E1 23791.547,E2 23791.547} C_VEL
LIN {X 0,Y 137.332,Z 760.298,A -85,B 0,C 180,E1 23804.222,E2 23804.222} C_VEL
LIN {X 0,Y 120.914,Z 769.784,A -85,B 0,C 180,E1 23819.941,E2 23819.941} C_VEL
LIN {X 0,Y 114.035,Z 774.01,A -85,B 0,C 180,E1 23834.6,E2 23834.6} C_VEL
LIN {X 0,Y 112.638,Z 775.378,A -85,B 0,C 180,E1 23850,E2 23850} C_VEL
LIN {X 0,Y 112.689,Z 774.97,A -85,B 0,C 180,E1 23858.139,E2 23858.139} C_VEL
LIN {X 0,Y 110.444,Z 773.898,A -85,B 0,C 180,E1 23867.025,E2 23867.025} C_VEL
LIN {X 0,Y 110.271,Z 772.024,A -85,B 0,C 180,E1 23876.121,E2 23876.121} C_VEL
LIN {X 0,Y 125.306,Z 764.052,A -85,B 0,C 180,E1 23893.543,E2 23893.543} C_VEL
LIN {X 0,Y 148.889,Z 750.657,A -85,B 0,C 180,E1 23907.034,E2 23907.034} C_VEL
LIN {X 0,Y 179.088,Z 730.331,A -85,B 0,C 180,E1 23916.846,E2 23916.846} C_VEL
LIN {X 0,Y 208.409,Z 706.039,A -85,B 0,C 180,E1 23922.985,E2 23922.985} C_VEL
LIN {X 0,Y 235.911,Z 677.616,A -85,B 0,C 180,E1 23927.12,E2 23927.12} C_VEL
LIN {X 0,Y 242.045,Z 670.298,A -85,B 0,C 180,E1 23927.883,E2 23927.883} C_VEL
LIN {X 0,Y 243.555,Z 666.301,A -85,B 0,C 180,E1 23931.061,E2 23931.061} C_VEL
LIN {X 0,Y 244.793,Z 662.877,A -85,B 0,C 180,E1 23936.456,E2 23936.456} C_VEL
LIN {X 0,Y 244.797,Z 663.045,A -85,B 0,C 180,E1 23940.002,E2 23940.002} C_VEL
LIN {X 0,Y 243.047,Z 668.236,A -85,B 0,C 180,E1 23946.259,E2 23946.259} C_VEL
LIN {X 0,Y 242.515,Z 670.056,A -85,B 0,C 180,E1 23947.693,E2 23947.693} C_VEL
LIN {X 0,Y 238.687,Z 674.945,A -85,B 0,C 180,E1 23948.506,E2 23948.506} C_VEL
LIN {X 0,Y 210.946,Z 704.862,A -85,B 0,C 180,E1 23952.554,E2 23952.554} C_VEL
LIN {X 0,Y 181.716,Z 730.465,A -85,B 0,C 180,E1 23958.591,E2 23958.591} C_VEL
LIN {X 0,Y 153.337,Z 751.065,A -85,B 0,C 180,E1 23967.288,E2 23967.288} C_VEL
LIN {X 0,Y 128.978,Z 766.509,A -85,B 0,C 180,E1 23979.813,E2 23979.813} C_VEL
LIN {X 0,Y 111.775,Z 776.954,A -85,B 0,C 180,E1 23997.19,E2 23997.19} C_VEL
LIN {X 0,Y 105.324,Z 781.651,A -85,B 0,C 180,E1 24013.29,E2 24013.29} C_VEL
LIN {X 0,Y 104.603,Z 783.278,A -85,B 0,C 180,E1 24030,E2 24030} C_VEL
LIN {X 0,Y 105.323,Z 781.672,A -85,B 0,C 180,E1 24046.71,E2 24046.71} C_VEL
LIN {X 0,Y 113.682,Z 775.772,A -85,B 0,C 180,E1 24065.585,E2 24065.585} C_VEL
LIN {X 0,Y 132.997,Z 764.046,A -85,B 0,C 180,E1 24082.838,E2 24082.838} C_VEL
LIN {X 0,Y 159.699,Z 746.826,A -85,B 0,C 180,E1 24095.018,E2 24095.018} C_VEL
LIN {X 0,Y 188.08,Z 725.458,A -85,B 0,C 180,E1 24102.939,E2 24102.939} C_VEL
LIN {X 0,Y 218.19,Z 697.92,A -85,B 0,C 180,E1 24108.581,E2 24108.581} C_VEL
LIN {X 0,Y 241.643,Z 671.667,A -85,B 0,C 180,E1 24111.834,E2 24111.834} C_VEL
LIN {X 0,Y 242.837,Z 669.498,A -85,B 0,C 180,E1 24112.835,E2 24112.835} C_VEL
LIN {X 0,Y 244.436,Z 664.297,A -85,B 0,C 180,E1 24118.223,E2 24118.223} C_VEL
LIN {X 0,Y 244.872,Z 663.26,A -85,B 0,C 180,E1 24119.998,E2 24119.998} C_VEL
LIN {X 0,Y 244.782,Z 663.21,A -85,B 0,C 180,E1 24123.544,E2 24123.544} C_VEL
LIN {X 0,Y 243.504,Z 666.996,A -85,B 0,C 180,E1 24129.41,E2 24129.41} C_VEL
LIN {X 0,Y 242.013,Z 670.579,A -85,B 0,C 180,E1 24132.024,E2 24132.024} C_VEL
LIN {X 0,Y 215.015,Z 700.015,A -85,B 0,C 180,E1 24135.852,E2 24135.852} C_VEL
LIN {X 0,Y 185.534,Z 725.585,A -85,B 0,C 180,E1 24141.511,E2 24141.511} C_VEL
LIN {X 0,Y 156.955,Z 745.73,A -85,B 0,C 180,E1 24149.747,E2 24149.747} C_VEL
LIN {X 0,Y 129.664,Z 761.732,A -85,B 0,C 180,E1 24163.127,E2 24163.127} C_VEL
LIN {X 0,Y 111.877,Z 771.238,A -85,B 0,C 180,E1 24181.082,E2 24181.082} C_VEL
LIN {X 0,Y 104.803,Z 775.339,A -85,B 0,C 180,E1 24201.693,E2 24201.693} C_VEL
LIN {X 0,Y 104.741,Z 775.665,A -85,B 0,C 180,E1 24210,E2 24210} C_VEL
LIN {X 0,Y 106.377,Z 774.261,A -85,B 0,C 180,E1 24226.539,E2 24226.539} C_VEL
LIN {X 0,Y 110.271,Z 772.024,A -85,B 0,C 180,E1 24236.121,E2 24236.121} C_VEL
LIN {X 0,Y 112.113,Z 769.41,A -85,B 0,C 180,E1 24245.015,E2 24245.015} C_VEL
LIN {X 0,Y 116.125,Z 766.033,A -85,B 0,C 180,E1 24253.468,E2 24253.468} C_VEL
LIN {X 0,Y 141.91,Z 752.484,A -85,B 0,C 180,E1 24268.603,E2 24268.603} C_VEL
LIN {X 0,Y 172.905,Z 732.919,A -85,B 0,C 180,E1 24278.503,E2 24278.503} C_VEL
LIN {X 0,Y 204.016,Z 708.374,A -85,B 0,C 180,E1 24284.757,E2 24284.757} C_VEL
LIN {X 0,Y 233.598,Z 678.773,A -85,B 0,C 180,E1 24288.939,E2 24288.939} C_VEL
LIN {X 0,Y 237.645,Z 673.96,A -85,B 0,C 180,E1 24289.498,E2 24289.498} C_VEL
LIN {X 0,Y 238.802,Z 670.999,A -85,B 0,C 180,E1 24292.718,E2 24292.718} C_VEL
LIN {X 0,Y 239.707,Z 669.07,A -85,B 0,C 180,E1 24296.381,E2 24296.381} C_VEL
LIN {X 0,Y 239.729,Z 669.208,A -85,B 0,C 180,E1 24300.002,E2 24300.002} C_VEL
LIN {X 0,Y 237.613,Z 674.361,A -85,B 0,C 180,E1 24306.264,E2 24306.264} C_VEL
LIN {X 0,Y 232.376,Z 680.777,A -85,B 0,C 180,E1 24307.206,E2 24307.206} C_VEL
LIN {X 0,Y 203.104,Z 710.368,A -85,B 0,C 180,E1 24311.389,E2 24311.389} C_VEL
LIN {X 0,Y 171.626,Z 735.881,A -85,B 0,C 180,E1 24317.874,E2 24317.874} C_VEL
LIN {X 0,Y 141.173,Z 756.076,A -85,B 0,C 180,E1 24327.768,E2 24327.768} C_VEL
LIN {X 0,Y 114.966,Z 771.115,A -85,B 0,C 180,E1 24343.584,E2 24343.584} C_VEL
LIN {X 0,Y 100.511,Z 779.394,A -85,B 0,C 180,E1 24363.132,E2 24363.132} C_VEL
LIN {X 0,Y 96.433,Z 782.559,A -85,B 0,C 180,E1 24380.966,E2 24380.966} C_VEL
LIN {X 0,Y 96.674,Z 782.99,A -85,B 0,C 180,E1 24390,E2 24390} C_VEL
LIN {X 0,Y 97.629,Z 781.378,A -85,B 0,C 180,E1 24408.07,E2 24408.07} C_VEL
LIN {X 0,Y 106.922,Z 775.583,A -85,B 0,C 180,E1 24427.885,E2 24427.885} C_VEL
LIN {X 0,Y 128.172,Z 763.743,A -85,B 0,C 180,E1 24445.785,E2 24445.785} C_VEL
LIN {X 0,Y 156.985,Z 746.122,A -85,B 0,C 180,E1 24457.957,E2 24457.957} C_VEL
LIN {X 0,Y 187.504,Z 723.783,A -85,B 0,C 180,E1 24465.703,E2 24465.703} C_VEL
LIN {X 0,Y 216.713,Z 697.573,A -85,B 0,C 180,E1 24470.712,E2 24470.712} C_VEL
LIN {X 0,Y 237.608,Z 674.766,A -85,B 0,C 180,E1 24473.53,E2 24473.53} C_VEL
LIN {X 0,Y 239.799,Z 669.42,A -85,B 0,C 180,E1 24479.998,E2 24479.998} C_VEL
LIN {X 0,Y 239.69,Z 669.394,A -85,B 0,C 180,E1 24483.619,E2 24483.619} C_VEL
LIN {X 0,Y 237.878,Z 673.694,A -85,B 0,C 180,E1 24489.997,E2 24489.997} C_VEL
LIN {X 0,Y 235.551,Z 676.732,A -85,B 0,C 180,E1 24490.748,E2 24490.748} C_VEL
LIN {X 0,Y 206.658,Z 706.147,A -85,B 0,C 180,E1 24494.733,E2 24494.733} C_VEL
LIN {X 0,Y 176.006,Z 730.84,A -85,B 0,C 180,E1 24500.683,E2 24500.683} C_VEL
LIN {X 0,Y 144.57,Z 751.103,A -85,B 0,C 180,E1 24510.225,E2 24510.225} C_VEL
LIN {X 0,Y 119.266,Z 764.575,A -85,B 0,C 180,E1 24523.931,E2 24523.931} C_VEL
LIN {X 0,Y 102.205,Z 772.843,A -85,B 0,C 180,E1 24543.613,E2 24543.613} C_VEL
LIN {X 0,Y 96.949,Z 775.628,A -85,B 0,C 180,E1 24561.015,E2 24561.015} C_VEL
LIN {X 0,Y 96.829,Z 775.953,A -85,B 0,C 180,E1 24570,E2 24570} C_VEL
LIN {X 0,Y 98.75,Z 774.552,A -85,B 0,C 180,E1 24587.858,E2 24587.858} C_VEL
LIN {X 0,Y 110.521,Z 768.805,A -85,B 0,C 180,E1 24608.061,E2 24608.061} C_VEL
LIN {X 0,Y 116.125,Z 766.033,A -85,B 0,C 180,E1 24613.468,E2 24613.468} C_VEL
LIN {X 0,Y 122.069,Z 761.934,A -85,B 0,C 180,E1 24621.166,E2 24621.166} C_VEL
LIN {X 0,Y 129.763,Z 757.086,A -85,B 0,C 180,E1 24628.01,E2 24628.01} C_VEL
LIN {X 0,Y 162.124,Z 738.533,A -85,B 0,C 180,E1 24639.057,E2 24639.057} C_VEL
LIN {X 0,Y 193.483,Z 715.868,A -85,B 0,C 180,E1 24645.565,E2 24645.565} C_VEL
LIN {X 0,Y 223.645,Z 688.262,A -85,B 0,C 180,E1 24649.89,E2 24649.89} C_VEL
LIN {X 0,Y 232.788,Z 678.424,A -85,B 0,C 180,E1 24651.009,E2 24651.009} C_VEL
LIN {X 0,Y 234.337,Z 675.062,A -85,B 0,C 180,E1 24656.298,E2 24656.298} C_VEL
LIN {X 0,Y 234.39,Z 675.165,A -85,B 0,C 180,E1 24660.002,E2 24660.002} C_VEL
LIN {X 0,Y 232.654,Z 678.995,A -85,B 0,C 180,E1 24664.958,E2 24664.958} C_VEL
LIN {X 0,Y 201.059,Z 710.53,A -85,B 0,C 180,E1 24669.181,E2 24669.181} C_VEL
LIN {X 0,Y 168.917,Z 735.807,A -85,B 0,C 180,E1 24675.292,E2 24675.292} C_VEL
LIN {X 0,Y 137.509,Z 755.772,A -85,B 0,C 180,E1 24684.711,E2 24684.711} C_VEL
LIN {X 0,Y 109.431,Z 770.814,A -85,B 0,C 180,E1 24700.447,E2 24700.447} C_VEL
LIN {X 0,Y 93.325,Z 779.097,A -85,B 0,C 180,E1 24720.874,E2 24720.874} C_VEL
LIN {X 0,Y 88.544,Z 782.268,A -85,B 0,C 180,E1 24740.154,E2 24740.154} C_VEL
LIN {X 0,Y 88.743,Z 782.701,A -85,B 0,C 180,E1 24750,E2 24750} C_VEL
LIN {X 0,Y 90.004,Z 781.086,A -85,B 0,C 180,E1 24769.661,E2 24769.661} C_VEL
LIN {X 0,Y 101.252,Z 774.94,A -85,B 0,C 180,E1 24791.609,E2 24791.609} C_VEL
LIN {X 0,Y 123.713,Z 763.443,A -85,B 0,C 180,E1 24808.952,E2 24808.952} C_VEL
LIN {X 0,Y 152.263,Z 746.966,A -85,B 0,C 180,E1 24820.283,E2 24820.283} C_VEL
LIN {X 0,Y 183.928,Z 724.817,A -85,B 0,C 180,E1 24827.842,E2 24827.842} C_VEL
LIN {X 0,Y 213.749,Z 699.011,A -85,B 0,C 180,E1 24832.62,E2 24832.62} C_VEL
LIN {X 0,Y 231.889,Z 680.214,A -85,B 0,C 180,E1 24834.834,E2 24834.834} C_VEL
LIN {X 0,Y 233.209,Z 677.992,A -85,B 0,C 180,E1 24836.276,E2 24836.276} C_VEL
LIN {X 0,Y 234.454,Z 675.371,A -85,B 0,C 180,E1 24839.998,E2 24839.998} C_VEL
LIN {X 0,Y 234.314,Z 675.377,A -85,B 0,C 180,E1 24843.702,E2 24843.702} C_VEL
LIN {X 0,Y 232.463,Z 679.111,A -85,B 0,C 180,E1 24849.035,E2 24849.035} C_VEL
LIN {X 0,Y 201.806,Z 709.082,A -85,B 0,C 180,E1 24853.004,E2 24853.004} C_VEL
LIN {X 0,Y 170.074,Z 733.392,A -85,B 0,C 180,E1 24858.93,E2 24858.93} C_VEL
LIN {X 0,Y 137.792,Z 752.911,A -85,B 0,C 180,E1 24868.468,E2 24868.468} C_VEL
LIN {X 0,Y 111.364,Z 765.97,A -85,B 0,C 180,E1 24882.816,E2 24882.816} C_VEL
LIN {X 0,Y 95.092,Z 773.134,A -85,B 0,C 180,E1 24901.466,E2 24901.466} C_VEL
LIN {X 0,Y 89.115,Z 775.916,A -85,B 0,C 180,E1 24920.218,E2 24920.218} C_VEL
LIN {X 0,Y 88.929,Z 776.24,A -85,B 0,C 180,E1 24930,E2 24930} C_VEL
LIN {X 0,Y 91.199,Z 774.842,A -85,B 0,C 180,E1 24949.393,E2 24949.393} C_VEL
LIN {X 0,Y 104.292,Z 769.097,A -85,B 0,C 180,E1 24970.793,E2 24970.793} C_VEL
LIN {X 0,Y 129.763,Z 757.086,A -85,B 0,C 180,E1 24988.01,E2 24988.01} C_VEL
LIN {X 0,Y 138.842,Z 751.653,A -85,B 0,C 180,E1 24993.994,E2 24993.994} C_VEL
LIN {X 0,Y 148.843,Z 745.136,A -85,B 0,C 180,E1 24999.119,E2 24999.119} C_VEL
